(* CoDeSys 2.3 library: Flexlink V2_0.lib *)
(* Libraries: TcUtilities.lib*3.2.16 16:08:58, TcSystem.lib*24.2.16 14:35:18, TcBase.lib 14.5.09 12:14:08, STANDARD.LIB 5.6.98 12:03:02, TcEtherCAT.lib 1.12.15 17:38:26 *)

(* Global variable list: Global_Variables *)
VAR_GLOBAL
(**************************************************************************************************************)
(* System Bit *)
(**************************************************************************************************************)

	OFF_50ms		: BOOL;
	ON_50ms		: BOOL;
	Clock50msOnPls	: BOOL;
	OFF_100ms		: BOOL;
	ON_100ms		: BOOL;
	Clock100msOnPls	: BOOL;
	OFF_500ms		: BOOL;
	ON_500ms		: BOOL;
	Clock500msOnPls	: BOOL;
	OFF_1s			: BOOL;
	ON_1s			: BOOL;
	Clock1sOnPls	: BOOL;
	Always_ON		:BOOL;
	Always_Off		:BOOL;
	Debug			:BOOL := TRUE;

(**************************************************************************************************************)
(* Machine Standard Word *)
(**************************************************************************************************************)

	ErrorDWord 			AT %MD1000:  ARRAY [0..20,1..10] OF DWORD;
	WarningDWord		AT%MD2000: ARRAY [0..20,1..10] OF DWORD;
	AutoDWord 			AT %MD3000:  ARRAY [0..20,1..10] OF DWORD;
	OriginDWord 			AT %MD4000:  ARRAY [0..20,1..10] OF DWORD;

	InputByte				AT %IB0: ARRAY [0..500] OF BYTE;
	OutputByte			AT %QB0: ARRAY [0..500] OF BYTE;

(**************************************************************************************************************)
(* Machine and Station Control *)
(**************************************************************************************************************)
	MC:Struc_Machine_Ctrl;
	SC :ARRAY[0..20] OF Struc_Station_Ctrl;

(**************************************************************************************************************)
(* Manual Control *)
(**************************************************************************************************************)
	ManualSafetyOK		:BOOL;
	M_StepFwdPls		:BOOL;
	M_StepBwdPls		:BOOL;
	M_StepRun			:BOOL;

(**************************************************************************************************************)
(* Input/Output *)
(**************************************************************************************************************)
	InputWord			AT%IB0	:ARRAY [0..100] OF BOOL;


END_VAR

(* Global variable list: Global_Variables_Error *)
VAR_GLOBAL
	E_EmgStop			: BOOL;
	E_LightCurtain		: BOOL;
	E_AirLow 			: BOOL;
	E_SafetyDoorOpen	: BOOL;
END_VAR

(* Global variable list: Global_Variables_HMI *)
VAR_GLOBAL
	T_AutoRunString:		STRING;

	T_StepRun:			BOOL;
	T_StepStop:			BOOL;
	T_StepBwd:			BOOL;
	T_StepFwd:			BOOL;
	T_StationError:		BOOL;
	T_Origin:				BOOL;
	T_OneCycleRun:		BOOL;
	T_ManualCycleTime:	TIME;
	T_Curr_Step_Station: 	UINT;
	T_EndProd:			BOOL;

	V_StepRunCurrStation:	STRING;
	V_StepRunStatus:		STRING;
	V_AutorunString:		STRING;
END_VAR

(* Global variable list: Global_Variables_Holding *)
VAR_GLOBAL RETAIN
	Password_Control: Std_Password_Ctrl;

(* Parameter Setting *)
	Number_of_Station : INT;

END_VAR

(* Data type *)
TYPE E_IndradriveDriveState :
(
	DriveState_Mode_PM  := 0,
	DriveState_Mode_bb,
	DriveState_Mode_Ab,
	DriveState_Mode_AH,
	DriveState_Mode_AF,
	DriveState_Mode_FC,
	DriveState_Mode_PC,
	DriveState_Mode_Invalid
);
END_TYPE

(* Data type *)
TYPE E_IndradriveErrorCode :
(
	INDRADRIVE_NO_ERROR := 0,
	INDRADRIVE_INVALID_ADDRESS_VALUE,
	INDRADRIVE_INVALID_DATA_VALUE,
	INDRADRIVE_PARA_WRITE_ERROR,
	INDRADRIVE_PARA_READ_ERROR,

	INDRADRIVE_ERROR_UNKNOWN := 999
);
END_TYPE

(* Data type *)
TYPE E_IndradriveListIndex :
(
	LIST_INDEX_0  := 0,
	LIST_INDEX_1,
	LIST_INDEX_2,
	LIST_INDEX_3,
	LIST_INDEX_4,
	LIST_INDEX_5,
	LIST_INDEX_6,
	LIST_INDEX_7,
	LIST_INDEX_8,
	LIST_INDEX_9,
	LIST_INDEX_10,
	LIST_INDEX_11,
	LIST_INDEX_12,
	LIST_INDEX_13,
	LIST_INDEX_14,
	LIST_INDEX_15,
	LIST_INDEX_16,
	LIST_INDEX_17,
	LIST_INDEX_18,
	LIST_INDEX_19,
	LIST_INDEX_20,
	LIST_INDEX_21,
	LIST_INDEX_22,
	LIST_INDEX_23,
	LIST_INDEX_24,
	LIST_INDEX_25,
	LIST_INDEX_26,
	LIST_INDEX_27,
	LIST_INDEX_28,
	LIST_INDEX_29,
	LIST_INDEX_30,
	LIST_INDEX_31,
	LIST_INDEX_MAX
);
END_TYPE

(* Data type *)
TYPE E_IndradriveOpMode :
(
	OP_MODE_DCP  := 0,
	OP_MODE_POS_01,
	OP_MODE_MUX_01,
	OP_MODE_MUX_02,
	OP_MODE_PROCESS_CNTRL,
	OP_MODE_USER := 99
);
END_TYPE

(* Data type *)
TYPE ST_ChecksumConfig :
STRUCT
	arChecksumConfigList            :  ARRAY [0..LIST_INDEX_MAX] OF WORD;       (* Read / write S_0_0327, IDN list of checksum parameter *)
	wCheckSumExpected             : WORD;                                                                     (* Read / write S-0-0326, Parameter checksum *)
END_STRUCT
END_TYPE

(* Data type *)
TYPE st_Indradrive_DCP_input :
STRUCT
	wAntriebsstatuswort   			: WORD;
	wSignalstatuswort   			: WORD;
	diLageistwert		  			: DINT;
	diIstgeschwindigkeit  			: DINT;
	dwDiagnosenummer				: DWORD;
END_STRUCT
END_TYPE

(* Data type *)
TYPE st_Indradrive_DCP_output :
STRUCT
	wMastersteuerwort   			: WORD;
	wSignalsteuerwort   			: WORD;
	diPositioniersollwert  			: DINT;
	diPositioniergeschwindigkeit  	: DINT;
END_STRUCT
END_TYPE

(* Data type *)
TYPE st_Indradrive_DCP_using_MUX_8_input :
STRUCT
	wDriveStatusWord : WORD;        (* S-0-0135: Drive Status word*)
	stMUX_in                 : st_Indradrive_MUX_8_input; (* 8 Channel Multiplexer Input Structure *)
END_STRUCT
END_TYPE

(* Data type *)
TYPE st_Indradrive_DCP_using_MUX_8_output :
STRUCT
	wMasterControlWord  : WORD;        (* S-0-0134: Master Control Word*)
	stMUX_out               : st_Indradrive_MUX_8_output; (* 8 Channel Multiplexer Output Structure *)
END_STRUCT
END_TYPE

(* Data type *)
TYPE st_Indradrive_MUX_1_input :
STRUCT
(*Struktur der benötigten Multiplexparameter (Teil der Echtzeitkanal-Eingangsdaten*)
	uiIndexAdressing	: UINT;		(*S-0-0368*)
      	uiListIndexWrite		: UINT;		(*S-0-0362*)
      	uiListIndexRead		: UINT;		(*S-0-0366*)
      	diReadValue1		: DINT;		(*S-0-0364*)
END_STRUCT
END_TYPE

(* Data type *)
TYPE st_Indradrive_MUX_1_output :
STRUCT
(*Struktur der benötigten Multiplexparameter (Teil der Echtzeitkanal-Ausgangsdaten*)
	uiIndexAdressing		: UINT;		(*S-0-0368*)
	uiListIndexWrite		: UINT;		(*S-0-0362*)
       	uiListIndexRead		: UINT;		(*S-0-0366*)
       	diWriteValue1		: DINT;		(*S-0-0360*)
END_STRUCT
END_TYPE

(* Data type *)
TYPE st_Indradrive_MUX_8_input :
STRUCT
(*Struktur der benötigten Multiplexparameter (Teil der Echtzeitkanal-Eingangsdaten*)
	uiIndexAdressing	: UINT;            (*S-0-0368*)
      	uiListIndexWrite		: UINT;            (*S-0-0362*)
      	uiListIndexRead		: UINT;            (*S-0-0366*)
      	dwReadValue1		: DWORD;     (*S-0-0364*)
    	dwReadValue2 		: DWORD;     (*S-0-0480 *)
    	dwReadValue3 		: DWORD;     (*S-0-0481 *)
    	dwReadValue4 		: DWORD;     (*S-0-0482 *)
    	dwReadValue5 		: DWORD;     (*S-0-0483 *)
    	dwReadValue6 		: DWORD;     (*S-0-0484 *)
    	dwReadValue7 		: DWORD;     (*S-0-0485 *)
    	dwReadValue8 		: DWORD;     (*S-0-0486 *)
END_STRUCT
END_TYPE

(* Data type *)
TYPE st_Indradrive_MUX_8_output :
STRUCT
(*Struktur der benötigten Multiplexparameter (Teil der Echtzeitkanal-Ausgangsdaten*)
	uiIndexAdressing		 : UINT;		    (*S-0-0368*)
	uiListIndexWrite		        : UINT;		    (*S-0-0362*)
     	uiListIndexRead		        : UINT;		    (*S-0-0366*)
      	dwWriteValue1                 : DWORD;      (*S-0-0360*)
	dwWriteValue2                 : DWORD;      (*S-0-0450 *)
	dwWriteValue3                 : DWORD;      (*S-0-0451 *)
	dwWriteValue4                 : DWORD;      (*S-0-0452 *)
	dwWriteValue5                 : DWORD;      (*S-0-0453 *)
	dwWriteValue6                 : DWORD;      (*S-0-0454 *)
	dwWriteValue7                 : DWORD;      (*S-0-0455 *)
	dwWriteValue8                 : DWORD;      (*S-0-0456 *)
END_STRUCT
END_TYPE

(* Data type *)
TYPE st_Indradrive_ProcessControl_input :
STRUCT
	wDriveStatusWord : WORD;                                                  (* S-0-0135: Drive Status word*)
	wSignalStatusWord : WORD;                                                (* S-0-0144: Singal Status word*)
	wProcessControlStatusWord : WORD;                              (* P-0-1410: Process Control status word coming from MLD program*)
	diVelocityAct : DINT;                                                                 (* S-0-0040: Actual velocity *)
	diPressureAct : DWORD;                                                               (* P-0-1372: Actual pressure value coming from MLD program  *)
	wAxisControllerMessage : WORD;                                      (*P-0-0555: Axis Controller Messages *)
	dwDriveDiagnosticNumber : DWORD;                               (* S-0-0390: Drive Diagnostic number *)
	diFlowAct :DWORD; 							    (* S-0-1301: Actual flow *)
	diAxisControllerMessage:WORD; 				    (*P-0-0555 Axis controller message*)
END_STRUCT
END_TYPE

(* Data type *)
TYPE st_Indradrive_ProcessControl_MUX_input :
STRUCT
	wDriveStatusWord : WORD;        (* S-0-0135: Drive Status word*)
	stMUX_in                 : st_Indradrive_MUX_8_input; (* 8 Channel Multiplexer Input Structure *)
END_STRUCT
END_TYPE

(* Data type *)
TYPE st_Indradrive_ProcessControl_MUX_output :
STRUCT
	wMasterControlWord  : WORD;        (* S-0-0134: Master Control Word*)
	stMUX_out               : st_Indradrive_MUX_8_output; (* 8 Channel Multiplexer Output Structure *)
END_STRUCT
END_TYPE

(* Data type *)
TYPE st_Indradrive_ProcessControl_output :
STRUCT
	wMasterControlWord  : WORD;          (* S-0-0134: Master Control Word*)
	wSignalControlWord : WORD;            (* S-0-0145: Signal Control Word*)
	wProcessControlWord : WORD;        (* P-0-1390: Process Control, Control Word, going to MLD Program *)
	diVelocityCmd : DINT;                            (* S-0-0036: Velocity Command value *)
	diPressureCmd : DINT;                          (* P-0-1371:Pressure Command value going to MLD Program *)
	diVolumePump01:DWORD; (**)
	diVolumePump02:DWORD;
	diVelocityLimitPos : DINT;                     (* P-0-1377:Postive Velocity Limit going to MLD Program *)
END_STRUCT
END_TYPE

(* Data type *)
TYPE Struc_Hist_Step_Case :
STRUCT
	CurrentStepHist	: INT;
	NextStepHist		: INT;
	StepTime		: TIME;
END_STRUCT
END_TYPE

(* Data type *)
TYPE Struc_Machine_Ctrl :
STRUCT
(* Mode Bit*)
	AutoMode		:BOOL;
	ManualMode		:BOOL;

(* Status Bit*)
	DryRun			:BOOL;
	Stop			:BOOL;
	AutoRunning		:BOOL;
	StopPressed		:BOOL;


	StationStopErr 	:BOOL;
	Warning			:BOOL;
	WarningBuzzer	:BOOL;
	Trouble			:BOOL;
	ErrDetection		:BOOL;


	OriginSchRun		:BOOL;
	InxOrigin			:BOOL;
	AllOrigin			:BOOL;
	AllStationRdy		:BOOL;
	AllStationNoWP 	:BOOL;

END_STRUCT
END_TYPE

(* Data type *)
TYPE Struc_Station_Ctrl :
STRUCT

	Running			:BOOL;
	AutoRun			:BOOL;
	RunReq			:BOOL;		(*Station Start Work Request*)
	Done			:BOOL;		(*Station Work Complete*)
	RunCond		:BOOL;
	Run_NextStepPls	:BOOL;
	Run_PrevStepPls	:BOOL;
	M_Step			:BOOL;

	Origin			:BOOL;   		(* Station Already Origin *)
	Rdy				:BOOL;		(* Station Ready *)
	NoWP 			:BOOL;
	MajorFault		:BOOL;		(* Station Major Fault *)
	MinorFault		:BOOL;		(* Station Minor Fault *)
	Warning			:BOOL;		(* Station Warning *)
	Bypass			:BOOL;		(* Station Bypass *)
	OriginSchRun		:BOOL;		(* Request Station to Origin *)

	Name			:STRING;
	Status			:STRING;
	CycleTime		:TIME;

END_STRUCT
END_TYPE

(* Data type *)
TYPE structIndradrive :
STRUCT
	In_ServoOn:BOOL;
	In_JogFwd:BOOL;
	In_JogBwd:BOOL;
	In_MoveHome:BOOL;
	In_SetAbsRef:BOOL;
	In_MoveAbs:BOOL;
	In_MoveRel:BOOL;
	In_StopMove:BOOL;
	In_VelCmd:REAL;
	In_PosCmd:REAL;
	In_MoveXLock:BOOL;	(*Mechanical Interlock*)
	Out_Ready:BOOL;
	Out_Busy:BOOL;
	Out_InPos:BOOL;
	Out_Referenced:BOOL;
	Out_PosLimit:BOOL;	(*1=OK*)
	Out_NegLimit:BOOL;	(*1=OK*)
	Out_Error:BOOL;
	Out_Warning:BOOL;
	Out_ErrorWord:WORD;
	Out_CurrPos:REAL;
	Out_CurrVel:REAL;
	Out_PosDirc:BOOL;	(*Moving in Positive Direction*)
	Out_NegDirc:BOOL;	(*Moving in Negative Direction*)
END_STRUCT
END_TYPE

(* POU Password_Output, ST *)
PROGRAM Password_Output
VAR

	pls_PasswordOK: R_TRIG;
	PasswordOKPls:BOOL;
END_VAR
(**************************************************************************************************************)
(* HMI Password Control*)
(**************************************************************************************************************)

Password_Control(
	In_PasswordConfig:= '9999');

pls_PasswordOK(CLK:= Password_Control.Out_PasswordOK OR Password_Control.Out_PasswordChanged);
PasswordOKPls := pls_PasswordOK.Q;

IF PasswordOKPls THEN
	CurrentVisu := 'TP40_SETTING';
END_IF
END_PROGRAM

(* POU Std_System_Out, LD *)
PROGRAM Std_System_Out
VAR

	Clk50ms:TON;
	ClkOff50ms:TON;
	Clk100ms:TON;
	ClkOff100ms:TON;
	Clk500ms:TON;
	ClkOff500ms:TON;
	ClkOn1s:TON;
	ClkOff1s:TON;

	T50ms_RTRIG: R_TRIG;
	T100ms_RTRIG: R_TRIG;
	T500ms_RTRIG: R_TRIG;
	T1s_RTRIG: R_TRIG;

END_VAR
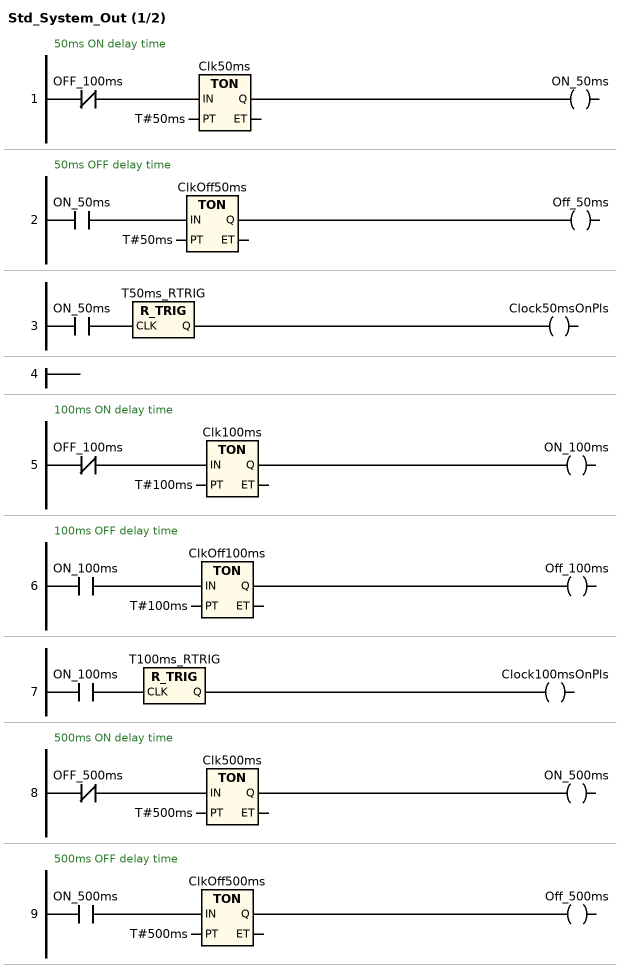
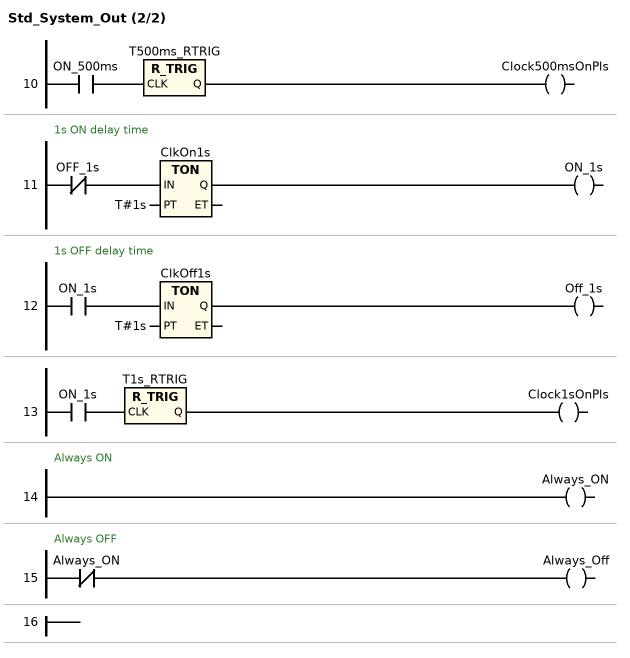
_LD_ (* Ladder Diagram *)
NETWORK 1 (* 50ms ON delay time *)
	[/OFF_100ms] - Clk50ms:TON(IN: *, PT: T#50ms) --- (ON_50ms)
NETWORK 2 (* 50ms OFF delay time *)
	[ON_50ms] - ClkOff50ms:TON(IN: *, PT: T#50ms) --- (Off_50ms)
NETWORK 3
	[ON_50ms] - T50ms_RTRIG:R_TRIG(CLK: *) --- (Clock50msOnPls)
NETWORK 4
	*
NETWORK 5 (* 100ms ON delay time *)
	[/OFF_100ms] - Clk100ms:TON(IN: *, PT: T#100ms) --- (ON_100ms)
NETWORK 6 (* 100ms OFF delay time *)
	[ON_100ms] - ClkOff100ms:TON(IN: *, PT: T#100ms) --- (Off_100ms)
NETWORK 7
	[ON_100ms] - T100ms_RTRIG:R_TRIG(CLK: *) --- (Clock100msOnPls)
NETWORK 8 (* 500ms ON delay time *)
	[/OFF_500ms] - Clk500ms:TON(IN: *, PT: T#500ms) --- (ON_500ms)
NETWORK 9 (* 500ms OFF delay time *)
	[ON_500ms] - ClkOff500ms:TON(IN: *, PT: T#500ms) --- (Off_500ms)
NETWORK 10
	[ON_500ms] - T500ms_RTRIG:R_TRIG(CLK: *) --- (Clock500msOnPls)
NETWORK 11 (* 1s ON delay time *)
	[/OFF_1s] - ClkOn1s:TON(IN: *, PT: T#1s) --- (ON_1s)
NETWORK 12 (* 1s OFF delay time *)
	[ON_1s] - ClkOff1s:TON(IN: *, PT: T#1s) --- (Off_1s)
NETWORK 13
	[ON_1s] - T1s_RTRIG:R_TRIG(CLK: *) --- (Clock1sOnPls)
NETWORK 14 (* Always ON *)
	* --- (Always_ON)
NETWORK 15 (* Always OFF *)
	[/Always_ON] --- (Always_Off)
NETWORK 16
	*
_END_LD_
(* the same logic as Structured Text *)
(* Network 1: 50ms ON delay time *)
Clk50ms(IN := NOT OFF_100ms, PT := T#50ms);
ON_50ms := Clk50ms.Q;
(* Network 2: 50ms OFF delay time *)
ClkOff50ms(IN := ON_50ms, PT := T#50ms);
Off_50ms := ClkOff50ms.Q;
(* Network 3 *)
T50ms_RTRIG(CLK := ON_50ms);
Clock50msOnPls := T50ms_RTRIG.Q;
(* Network 4 *)
(* Network 5: 100ms ON delay time *)
Clk100ms(IN := NOT OFF_100ms, PT := T#100ms);
ON_100ms := Clk100ms.Q;
(* Network 6: 100ms OFF delay time *)
ClkOff100ms(IN := ON_100ms, PT := T#100ms);
Off_100ms := ClkOff100ms.Q;
(* Network 7 *)
T100ms_RTRIG(CLK := ON_100ms);
Clock100msOnPls := T100ms_RTRIG.Q;
(* Network 8: 500ms ON delay time *)
Clk500ms(IN := NOT OFF_500ms, PT := T#500ms);
ON_500ms := Clk500ms.Q;
(* Network 9: 500ms OFF delay time *)
ClkOff500ms(IN := ON_500ms, PT := T#500ms);
Off_500ms := ClkOff500ms.Q;
(* Network 10 *)
T500ms_RTRIG(CLK := ON_500ms);
Clock500msOnPls := T500ms_RTRIG.Q;
(* Network 11: 1s ON delay time *)
ClkOn1s(IN := NOT OFF_1s, PT := T#1s);
ON_1s := ClkOn1s.Q;
(* Network 12: 1s OFF delay time *)
ClkOff1s(IN := ON_1s, PT := T#1s);
Off_1s := ClkOff1s.Q;
(* Network 13 *)
T1s_RTRIG(CLK := ON_1s);
Clock1sOnPls := T1s_RTRIG.Q;
(* Network 14: Always ON *)
Always_ON := TRUE;
(* Network 15: Always OFF *)
Always_Off := NOT Always_ON;
(* Network 16 *)
END_PROGRAM

(* POU F_GetVersionDC_IA_Indradrive, ST *)
FUNCTION F_GetVersionDC_IA_Indradrive : UINT
VAR_INPUT
       nVersionElement       :       INT;
END_VAR 
VAR
END_VAR
(* Version history:
Date               | Version  | created under             | Author            | Remark 
------------------------------------------------------------------------------------------------------------------------------------------------------------------------------ 
03/01/2012    | 1.0.0      | V2.11.0 (Build 1514) | U. Chauhan   | first release 
------------------------------------------------------------------------------------------------------------------------------------------------------------------------------ 
20/08/2012    | 1.1.0      | V2.11.0 (Build 1514) | U. Chauhan   | 
	Old Process Control FB is renamed as Process control using MUX Version 1.0. 
	New ProcessControl FB Version 1.0 without MUX added.
------------------------------------------------------------------------------------------------------------------------------------------------------------------------------ 
29/10/2012    | 1.1.1      | V2.11.0 (Build 1514) | U. Chauhan   | "Process Control FB" and "Process control using MUX FB"  updated to Version 1.1
	DriveAH Bit added to both the FB and activated along with DriveStart Input.
11/12/2012    | 1.1.2      | V2.11.0 (Build 1514) | U. Chauhan   | "Process Control FB" updated to Version 1.2 and "Process control using MUX FB" updated to Version 1.2
	some bug fixes and calculations updated as per  
18/02/2013    | 1.2.0      | V2.11.0 (Build 1514) | U. Chauhan   | "Process Control FB" updated to Version 1.3 
	It is now possibile to use Pressure Value and Flowrate values in Percentage, 
	Selection of the Parameter Set is now possible with Input field
	FlowRateMaximum vlaue will be passed on to Drive as a positive Velocity Limit
05/08/2013    | 1.3.0      | V2.11.0 (Build 1514) | U. Chauhan   | SIP Implementation for Parameter Access added.
					FBs for Read Everything, ReadDescription, ReadOnlyData, ReadSegment, Read DataStatus,
					WriteData and WriteDatabits added.
------------------------------------------------------------------------------------------------------------------------------------------------------------------------------ 
26/02/2014    | 2.0.0      | V2.11.0 (Build 1514) | U. Chauhan   | SIPParameter Access FBs have been moved to another library due to license issues with TCPIP server. 
------------------------------------------------------------------------------------------------------------------------------------------------------------------------------ 
20.08.2014     |2.1.0	     | V2.11.0 (Build 1514) | Arun R            | FB_ProcessControl update of drive halt and flow rate decimal point logic. 
------------------------------------------------------------------------------------------------------------------------------------------------------------------------------ 
15/09/2014     |2.2.0	     | V2.11.0 (Build 1514) | Pradeep R           |  FB_Indradrive_DCP drive enable updated to stay on always to prevent torque free mode 
------------------------------------------------------------------------------------------------------------------------------------------------------------------------------ 
*) 

CASE nVersionElement OF
1: (* major number *)
       F_GetVersionDC_IA_Indradrive := 2;
2: (* minor number *)
       F_GetVersionDC_IA_Indradrive := 2;
3: (* revision number *)
       F_GetVersionDC_IA_Indradrive := 0;
ELSE
   F_GetVersionDC_IA_Indradrive := 16#FFFF;
END_CASE
END_FUNCTION

(* POU FB_ConfigChecksum, ST *)
(*#########################################################################################*)
(* General Header *)
(*----------------------------------------------------------------------------------------------------------------------------------------------------------------*)
(* Short description :		      Function Block for configuring & checking Checksum parameters in Indradrive              *)
(* Version : 					      01VRS                                                                                                                                       *)
(* Name : 					      Upendra Chauhan                                                                                                                    *)
(* Date : 					      2012-03-23                                                                                                                               *)
(* Company : 				      Bosch Rexroth AG                                                                                                                    *)
(* Target : 					      >MPx07VRS                                                                                                                             *)
(* Functional description :		With the help of this function block configurable Checksum feature of Indradrive            *)
(*                                                     User defined parameter list is at first written to paramter S-0-0327                            *)
(*                                                     This is enable the drive to calculate the checksum value for these parameter which is  *)
(*                                                     in turn written by Indradrive to Parameter S-0-0326                                                            *)
(*                                                     The FB reads this parameter anc compare is with Desired Checksum value as given *)
(*                                                     by user. If the value match the desired checksum good result is stored in  output           *)
(*                                                     bCheckSumOk. Actual checksum value is stored in dwActCheckSum and error Id is   *)
(*                                                     displayed in case of any error in dwErrorID                                                                         *)
(*----------------------------------------------------------------------------------------------------------------------------------------------------------------*)
(* Handling specials :                                                                                                                                                                      *)
(*----------------------------------------------------------------------------------------------------------------------------------------------------------------*)
(* Additional Header                                                                                                                                                                        *)
(*----------------------------------------------------------------------------------------------------------------------------------------------------------------*)
(* Version : 					 *)
(* Name : 					 *)
(* Date : 						 *)
(* Company : 					 *)
(* *)
(* *)
(* *)
(*-----------------------------------------------------------------------------------------------------------------------------------------------------------------*)
(*##########################################################################################*)
(*##########################################################################################*)
FUNCTION_BLOCK FB_ConfigChecksum
VAR_INPUT
	bExecute			 : BOOL;
	pstPlcDriveRef          : POINTER TO ST_PLCDriveRef;
	pstChecksumConfig : POINTER TO ST_ChecksumConfig;
END_VAR
(*___________________________________________________________________________________________________________________*)
(*___________________________________________________________________________________________________________________*)
VAR_OUTPUT
	bActive				: BOOL;										(*FB Active*)
	bDone                       : BOOL;
	bError				: BOOL;										(*Error in FB*)
	bCheckSumOk		: BOOL;										(*TRUE - Right config loaded / FALSE- Wrong Config*)
	dwActCheckSum     : DWORD := 0;                                                          (* Actual Checksum value, S-0-0326, Parameter checksum *)
	dwErrorID                 : DWORD := 0;                                                          (* Actual Checksum value, S-0-0326, Parameter checksum *)
END_VAR

VAR_IN_OUT
END_VAR
(*___________________________________________________________________________________________________________________*)
(*___________________________________________________________________________________________________________________*)
VAR
	stDriveRef                 : ST_DriveRef;
	iStep				: USINT;
	nElement 			: BYTE 				:=  64 ;					(*In case of list parameter the element of the list to be read or written*)
	bReadPar      		: BOOL 			:= FALSE;				(*command to read the parameter*)
	bReadErr       		: BOOL;										(*error in reading*)
	bWritePar			: BOOL;										(*command to write the parameter*)
	bWriteActive		: BOOL;										(*writing in progress*)
	bErrorWrite			: BOOL;										(*error in writing*)
	bWriteErr			: BOOL;										(*error in writing*)
	bReadActive		: BOOL;										(*reading in progress*)


	arConfigByteValue 	: ARRAY [0..100] OF BYTE;		     			(*array of bite values*)

 	 (*Function block declaration*)
	fbSercosParaWrite	: FB_SoEWrite_ByDriveRef;				(*write fb call*)
	fbSercosParaRead	: FB_SoERead_ByDriveRef;				(*read fb call*)
(*___________________________________________________________________________________________________________________*)
	iListIndex : INT := 0;
	wNoOfBytesTransfered: WORD;
	arbyReadValue : ARRAY [0..4] OF BYTE;
	R_TRIG_bExecute: R_TRIG;
END_VAR
(*___________________________________________________________________________________________________________________
Name of the Project			:CheckSumFBCode.pro
Name of the PLC System		:TWINCAT
Name of the DRIVE/Firmware	:Rexroth Indradrive HCS01.1E / 16VRS 
Version of Software used		:TwinCAT V2.11.0(Build 2209)
Version of Function Block		:V1.0
Author						: Upendra Chauhan
Date						:23.03.2012
___________________________________________________________________________________________________________________*)

(*FUNCTION BLOCK USED TO VERIFY THE CONFIGURATION FOR REXROTH INDRA DRIVE SETTINS ARE MADE CORRECTLY*)

(* rising edge at bExecute *)
R_TRIG_bExecute ( CLK := bExecute );

(* execute cycle *)
CASE iStep OF
	0:										(*WAIT FOR EXECUTE COMMAND*)
		 IF R_TRIG_bExecute.Q THEN
			bActive :=TRUE;
			dwActCheckSum := 0;                                                          (* Actual Checksum value, S-0-0326, Parameter checksum *)
			iStep:=1;
		 END_IF

		IF (bExecute = FALSE) THEN
			bDone :=FALSE;
			bError := FALSE;
			bCheckSumOk :=FALSE;
			dwErrorID := INDRADRIVE_NO_ERROR;
		 END_IF

	1:
		IF pstPlcDriveRef = 0 OR pstChecksumConfig = 0 THEN
			dwErrorID := INDRADRIVE_INVALID_ADDRESS_VALUE;
			iStep:=200;
		ELSE
			iStep:=5;
		END_IF

	5:
		stDriveRef.sNetId     := F_CreateAmsNetId(pstPlcDriveRef^.aNetId);
		stDriveRef.nSlaveAddr := pstPlcDriveRef^.nSlaveAddr;
		stDriveRef.nDriveNo   := pstPlcDriveRef^.nDriveNo;
		stDriveRef.nDriveType := pstPlcDriveRef^.nDriveType;
		IF (stDriveRef.sNetId <> '') AND (stDriveRef.nSlaveAddr <> 0) THEN
			iStep:= 10;
		ELSE
			dwErrorID := INDRADRIVE_INVALID_DATA_VALUE;
			iStep:= 200;
		END_IF

	10:
		FOR iListIndex := 0 TO LIST_INDEX_MAX DO
			IF  ( pstChecksumConfig^.arChecksumConfigList[iListIndex] = 0 )
			THEN
				IF iListIndex = 0 THEN
					(* if First two parameter are Zero then error exit *)
					IF ( pstChecksumConfig^.arChecksumConfigList[iListIndex + 1] = 0 ) THEN
						dwErrorID := INDRADRIVE_INVALID_DATA_VALUE;
						iStep:= 200;
						(* exit loop as list has invalid *)
						EXIT;
					END_IF
				ELSE
					(* if two consicutive parameter are Zero or Last list para is zero , the list is completed *)
					IF ( pstChecksumConfig^.arChecksumConfigList [iListIndex -1] = 0 ) OR
					    (  iListIndex = LIST_INDEX_MAX )
					THEN
						IF ( pstChecksumConfig^.arChecksumConfigList [iListIndex -1] = 0 )
						THEN
							(* reduce one step if last value was also zero *)
							iListIndex := iListIndex - 1;
						END_IF
						(* exit loop as list is completed *)
						EXIT;
					END_IF
				END_IF
			END_IF
		END_FOR

		(* Byte length = Number of words x 2 *)
		wNoOfBytesTransfered :=  iListIndex  * 2 ;

		(* first four values of arConfigByteValue depends on the number of Bytes to be transfered *)
		(* convert word value Maximum bytes to array of bytes *)
		MEMCPY ( ADR(arConfigByteValue), ADR(wNoOfBytesTransfered ), 2);
		(* convert word value Maximum bytes to array of bytes *)
		MEMSET ( ADR(arConfigByteValue[2]), 0, 2);
		(* convert wrod array to byte array *)
		MEMCPY ( ADR(arConfigByteValue[4]), ADR(pstChecksumConfig^.arChecksumConfigList), SIZEOF (pstChecksumConfig^.arChecksumConfigList));

		(* write S_0_0327, IDN list of checksum parameter *)
		bWritePar :=TRUE;

		iStep          :=15;

	15:										(*WAIT TILL WRITE bExecuteS*)
		IF bErrorWrite THEN
			(* error writing parameter to Indradrive *)
			dwErrorID := INDRADRIVE_PARA_WRITE_ERROR;
			bWritePar := FALSE;
			iStep:=200;
		ELSE
			IF( NOT bWriteActive ) THEN
				bWritePar := FALSE;
				iStep:=20;
			END_IF
		END_IF

	20:										(*READ THE S326 CHECKSUM VALUE PARAMETER*)
		bReadPar:=TRUE;
		iStep:=25;

	25:										(*WAIT TILL READ bExecuteS*)
		IF bReadErr THEN
			(* error reading parameter from Indradrive *)
			dwErrorID := INDRADRIVE_PARA_READ_ERROR;
			bReadPar:= FALSE;
			iStep:=200;
		ELSE
			IF( NOT bReadActive ) THEN
				bReadPar:= FALSE;
				iStep:=30;
			END_IF
		END_IF

	30:										(*CONVERT READ BYTE VALUE TO WORD VALUE*)
		(* copy read checksum  Byte array to word value *)
		MEMCPY (ADR (dwActCheckSum), ADR(arbyReadValue), 4);
		iStep:=35;

	35:										(*COMPARE WITH PREPROGRAMMED CHECKSUM VALUE TO VALIDATE RIGHT CONFIGURATION*)
		IF ( dwActCheckSum = pstChecksumConfig^.wCheckSumExpected) THEN
			bCheckSumOk :=TRUE;
		ELSE
			bCheckSumOk :=FALSE;
		END_IF
		iStep  :=40;

	40:										(*RESET FUNCTION BLOCK*)
		bDone :=TRUE;
		bActive:=FALSE;
		iStep:=0;

	200:									(*ERROR STEP*)
		bActive:=FALSE;
		bError := TRUE;
		iStep := 0;
END_CASE


(*Write fub function call*)
fbSercosParaWrite(
	stDriveREf := stDriveRef,
	nIdn:= 327 ,                                                            (* Parameter S-0-0327 : IDN list of checksum parameter *)
	nElement:= nElement  ,                                        (* Write 'Value' nElement := 0x40 *)
	pSrcBuf:=ADR (arConfigByteValue) ,
	cbBufLen:=SIZEOF(arConfigByteValue) ,
	bExecute:=bWritePar ,
	tTimeout:=T#10s,
	bBusy=>bWriteActive ,
	bError=>bWriteErr ,
	iAdsErrId=> ,
	 iSercosErrId => );

(*Read fub function call*)
fbSercosParaRead(
	stDriveREf := stDriveRef,
	nIdn:=326 ,                                                            (* Parameter S-0-0326 : checksum value *)
	nElement:=nElement ,                                         (* read 'Value' nElement := 0x40 *)
	pDstBuf:= ADR (arbyReadValue) ,
	cbBufLen:= SIZEOF(arbyReadValue) ,
	bExecute:=bReadPar ,
	tTimeout:=T#10s ,
	bBusy=>bReadActive	 ,
	bError=>bReadErr ,
	iAdsErrId=> ,
	iSercosErrId => ,
	dwAttribute => );
END_FUNCTION_BLOCK

(* POU FB_Indradrive_DCP, ST *)
(*############################################################################################*)
(* General Header *)
(*-----------------------------------------------------------------------------------------------------------------------------------------------------------------*)
(* Short description :			Funktionsbaustein „Antriebsgeführtes Positionieren“ über Ehtercat *)
(* Version : 					01VRS *)
(* Name : 					Michael Lippert *)
(* Date : 						2010-11-12*)
(* Company : 					BoschRexroth AG *)
(* Target : 					>MPx07VRS *)
(* Functional description :		Mit Hilfe dieses Funktionsbausteins „DCP_INDRADRIVE“ kann der Antrieb in der
								Betriebsart „Antriebsgeführtes Positionieren“ durch Vorgabe des S-0-0282,
								Positioniersollwert (POS_CMD) und des S-0-0259, Positioniergeschwindigkeit (VEL_CMD) 
								relativ oder absolut positioniert werden. Mit diesem Funktionsbaustein werden ferner 
								die Funktionen Tippen, Referenzieren und Fehler löschen angesteuert.
*)
(* Handling specials : *)
(*-----------------------------------------------------------------------------------------------------------------------------------------------------------------*)
(* Additional Header *)

(*------------------------------------------------------------------------------------------------------------------------------------------------------------------------*)
(* Version : 1.1.0	                                                                                                                                                                                              *)
(* Name : prd6kor ( DC-IA/EDY )                                                                                                                                                                   *)
(*Date: 15.09.2014                                                                                                                                                                                                *)
(* Company : Bosch Rexroth                                                                                                                                                                            *)
(* "FB_Indradrive_DCP" updated drive enable to prevent torque free mode on motor					                      *)
(*------------------------------------------------------------------------------------------------------------------------------------------------------------------------*)


(*############################################################################################*)
(*############################################################################################*)
FUNCTION_BLOCK FB_Indradrive_DCP
VAR_INPUT
     bDRIVE_ENABLE 					: BOOL; 						(*Antriebstatus Uebergang AB -> AH, Drive Enable state of drive change Ab->AH *)
     bDRIVE_START 					: BOOL; 						(*Antriebstatus Uebergang AH -> AF, Drive Enable state of drive change AH->AF *)
     bHOMING 							: BOOL; 						(*Achse Referenzieren, Homing the axis*)
     bRESET 							: BOOL; 						(*Stoerung quittieren, Reset Error*)
     bJOG_FORWARD 					: BOOL; 						(*Tippen vorwaerts, Jog forward*)
     bJOG_BACKWARD					: BOOL;						(*Tippen rueckwaerts, Jog backward*)
     bNEW_VALUE 						: BOOL; 						(*neuer Sollwert, new value *)
     bABS_REL 						: BOOL; 						(*Position Absolut = 0 oder Relativ = 1, position = absoluteor relative  *)
     bIMMEDIATE_CHANGE 				: BOOL; 						(*Satzsofortwechsel 1= sofort, immediate block change 1= immediately*)
     diPOS_CMD 						: DINT; 						(*Soll-Position, Command position*)
     diVEL_CMD 						: DINT; 						(*Soll-Geschwindigkeit, command velocity*)
     stEK_IN							: st_Indradrive_DCP_input;		(*Eingangsdaten (input data*)
END_VAR
VAR_OUTPUT
     bQ_DRIVE_ENABLE 				: BOOL; 						(*Quittierung DRIVE_ENABLE, acknowledge DRIVE_ENABLE*)
     bQ_MAIN_MODE 					: BOOL; 						(*Quittierung MAIN_MODE, acknowledge MAIN_MODE*)
     bIN_REFERENCE 					: BOOL; 						(*Referenziert, In_Reference*)
     bPOS_OK 							: BOOL; 						(*Sollwert erreicht = 1, target position reached = 1*)
     bNEW_VALUE_POSSIBLE 			: BOOL; 						(*Neuer Sollwert moeglich, NEW_VALUE_POSSIBLE*)
     bSTATUS_MESSAGE 				: BOOL; 						(*STATUS_MESSAGE*)
     bWARNING 						: BOOL; 						(*WARNING*)
     bERROR 							: BOOL; 						(*ERROR*)
     bIN_STANDSTILL 					: BOOL; 						(*IN_STANDSTILL*)
     dwDRIVE_DIAGNOSIS 				: DWORD; 					(*DRIVE_DIAGNOSIS*)
     diPOS_ACT 						: DINT; 						(*Aktuelle Position, actual position*)
     diVEL_ACT 						: DINT; 						(*Aktuelle Geschwindigkeit, actual velocity*)
     stEK_OUT 							: st_Indradrive_DCP_output;	(*Ausgangsdaten (output data*)
END_VAR
VAR
	bInternHalt 						: BOOL; 						(*INTERN_Halt*)
	bInternFrg 						: BOOL; 						(*INTERN_FRG*)
	bInternPosStart 					: BOOL; 						(*INTERN_POS_START*)
	bInternHoming 					: BOOL; 						(*INTERN_HOMING*)
	bInternJogForward 				: BOOL;						(*INTERN_JOG_FORWARD*)
	bInternJogBackward 				: BOOL; 						(*INTERN_JOG_BACKWARD*)
	bNewValueFlanke 				: BOOL; 						(*NEW_VALUE_FLANKE*)
	bNewValueImpulse 				: BOOL; 						(*NEW_VALUE_IMPULSE*)
END_VAR
(*###############################################################################*)
(*####  Bildung Statusbits Baustein									    	  ###*)
(*###############################################################################*)

(* Drive in AF? *)
bQ_DRIVE_ENABLE				:= stEK_IN.wAntriebsstatuswort.14
									AND stEK_IN.wAntriebsstatuswort.15;

(* Drive enabled (in AF) + Drive Follows Cmd + Primary OpMode active *)
bQ_MAIN_MODE 					:= stEK_IN.wAntriebsstatuswort.3
									AND bQ_DRIVE_ENABLE
									AND NOT stEK_IN.wAntriebsstatuswort.8
									AND NOT stEK_IN.wAntriebsstatuswort.9
									AND NOT stEK_IN.wAntriebsstatuswort.10;

bNEW_VALUE_POSSIBLE			:=   	stEK_OUT.wSignalsteuerwort.0 AND
									 stEK_IN.wSignalstatuswort.10 OR
									(
										NOT stEK_OUT.wSignalsteuerwort.0 AND
										NOT stEK_IN.wSignalstatuswort.10
									) AND
									stEK_IN.wAntriebsstatuswort.15 AND  (* actually redundant with bQ_MAIN_MODE *)
									bQ_MAIN_MODE AND
									bInternPosStart;

(*##################################################################################*)
(*####  Bildung interner Zuständsbits 											 ###*)
(*##################################################################################*)

bInternHoming 					:= bInternFrg AND NOT bInternPosStart AND NOT bJOG_FORWARD
									AND NOT bJOG_BACKWARD AND bHOMING;

bInternJogForward 				:= bInternFrg AND NOT bInternPosStart AND bJOG_FORWARD
									AND NOT bJOG_BACKWARD AND NOT bHOMING;

bInternJogBackward 				:= bInternFrg AND NOT bInternPosStart AND NOT bJOG_FORWARD
									AND bJOG_BACKWARD AND NOT bHOMING;

bInternPosStart					:= bInternFrg AND NOT bJOG_FORWARD
									AND NOT bJOG_BACKWARD AND NOT bHOMING;

bInternHalt						:= bDRIVE_ENABLE;

bInternFrg 						:= bInternHalt AND bQ_DRIVE_ENABLE AND bDRIVE_START;

(*##################################################################################*)
(*####  Bildung Togglebit für Sollwertübernahme 								 ###*)
(*##################################################################################*)

bNewValueImpulse				:= bNEW_VALUE AND NOT bNewValueFlanke;

bNewValueFlanke					:= bNEW_VALUE;

IF (bNEW_VALUE_POSSIBLE OR bIMMEDIATE_CHANGE) AND bInternPosStart AND bNewValueImpulse THEN
	stEK_OUT.diPositioniersollwert := diPOS_CMD;
	IF (stEK_IN.wSignalstatuswort.10 XOR stEK_OUT.wSignalsteuerwort.0) AND bIMMEDIATE_CHANGE THEN
		stEK_OUT.wSignalsteuerwort.0 := stEK_IN.wSignalstatuswort.10;
	ELSE
		stEK_OUT.wSignalsteuerwort.0 := NOT stEK_IN.wSignalstatuswort.10;
	END_IF
(*Verhinderung F2050 -->nicht nötig Anwenderfehler sollen zu Antriebsfehlern führen*)
(*ELSE
	IF stEK_IN.wAntriebsstatuswort.3
	OR (stEK_IN.wAntriebsstatuswort.8 OR stEK_IN.wAntriebsstatuswort.9 OR stEK_IN.wAntriebsstatuswort.10)
	AND bQ_DRIVE_ENABLE THEN
		stEK_OUT.wSignalsteuerwort.0 := stEK_IN.wSignalstatuswort.10;
	END_IF*)
END_IF


(*##################################################################################*)
(*#### Ausgabe auf zyklische Daten												 ###*)
(*##################################################################################*)

stEK_Out.wSignalsteuerwort.2			:= bInternHoming;
stEK_Out.wSignalsteuerwort.3			:= bABS_REL;
stEK_Out.wSignalsteuerwort.4			:= bIMMEDIATE_CHANGE;
stEK_Out.wSignalsteuerwort.5			:= bRESET;
stEK_Out.wSignalsteuerwort.6			:= bInternJogForward;
stEK_Out.wSignalsteuerwort.7			:= bInternJogBackward ;


stEK_OUT.wMastersteuerwort.13 		:= bInternFrg;


(*####   b.14 is made alwasy on to prevent torque free mode on servo						 ###*)
stEK_OUT.wMastersteuerwort.14 		:= TRUE;


stEK_OUT.wMastersteuerwort.15 		:= bInternHalt;


stEK_OUT.diPositioniergeschwindigkeit 	:= diVEL_CMD;


(*##################################################################################*)
(*#### Einlesen von zyklischen Daten											 ###*)
(*##################################################################################*)

diPOS_ACT 						:= stEK_IN.diLageistwert;
diVEL_ACT 						:= stEK_IN.diIstgeschwindigkeit;
dwDRIVE_DIAGNOSIS 			:= stEK_IN.dwDiagnosenummer;
bSTATUS_MESSAGE 				:= stEK_IN.wAntriebsstatuswort.11;
bWARNING 						:= stEK_IN.wAntriebsstatuswort.12;
bERROR 						:= stEK_IN.wAntriebsstatuswort.13;
bIN_REFERENCE 				:= stEK_IN.wSignalstatuswort.2;
bPOS_OK 						:= stEK_IN.wSignalstatuswort.4;
bIN_STANDSTILL 				:= stEK_IN.wSignalstatuswort.3;
END_FUNCTION_BLOCK

(* POU FB_Indradrive_DCP_using_MUX_8, ST *)
(*#########################################################################################*)
(* General Header *)
(*----------------------------------------------------------------------------------------------------------------------------------------------------------------*)
(* Short description :		      Function Block Drive Controlled positioning using Multiplex Channel“ over      Ethercat *)
(* Version : 					      01VRS                                                                                                                                       *)
(* Name : 					      Upendra Chauhan                                                                                                                    *)
(* Date : 					      2012-02-23                                                                                                                               *)
(* Company : 				      Bosch Rexroth AG                                                                                                                    *)
(* Target : 					      >MPx07VRS                                                                                                                             *)
(* Functional description :		With the help of this function block Indradrive can be used with Drive Contrlled              *)
(*                                                     Positioning mode. The Function block is same as                                                              *)
(*                                                     "FB_DCP_INDRADRIVE_EtherCAT_ST" except the cyclic data transmission.             *)
(*                                                     Here 8 Channel Multiplexer is used for cyclic data read and write. The index used is    *)
(*                                                     predefined as '0'. The required Parameter in AT are configured in Multiplex config list  *)
(*                                                     e.g. S-0-0370, S-0-0490 - S-0-0496 element number '0'                                                   *)
(*                                                     Similarly required MDT parameters are configured in config list S-0-0371, S-0-0500-  *)
(*                                                     S-0-0506 element number '0'                                                                                                 *)
(*----------------------------------------------------------------------------------------------------------------------------------------------------------------*)
(* Handling specials :                                                                                                                                                                      *)
(*----------------------------------------------------------------------------------------------------------------------------------------------------------------*)
(* Additional Header                                                                                                                                                                        *)
(*----------------------------------------------------------------------------------------------------------------------------------------------------------------*)
(* Version : 					 *)
(* Name : 					 *)
(* Date : 						 *)
(* Company : 					 *)
(* *)
(* *)
(* *)
(*-----------------------------------------------------------------------------------------------------------------------------------------------------------------*)
(*##########################################################################################*)
(*##########################################################################################*)
FUNCTION_BLOCK FB_Indradrive_DCP_using_MUX_8
VAR_INPUT
     bDRIVE_ENABLE 					: BOOL; 						(*Antriebstatus Uebergang AB -> AH, Drive Enable state of drive change Ab->AH *)
     bDRIVE_START 					: BOOL; 						(*Antriebstatus Uebergang AH -> AF, Drive Enable state of drive change AH->AF *)
     bHOMING 							: BOOL; 						(*Achse Referenzieren, Homing the axis*)
     bRESET 							: BOOL; 						(*Stoerung quittieren, Reset Error*)
     bJOG_FORWARD 					: BOOL; 						(*Tippen vorwaerts, Jog forward*)
     bJOG_BACKWARD					: BOOL;						(*Tippen rueckwaerts, Jog backward*)
     bNEW_VALUE 						: BOOL; 						(*neuer Sollwert, new value *)
     bABS_REL 						       : BOOL; 						(*Position Absolut = 0 oder Relativ = 1, position = absoluteor relative  *)
     bIMMEDIATE_CHANGE 				: BOOL; 						(*Satzsofortwechsel 1= sofort, immediate block change 1= immediately*)
     diPOS_CMD 						: DINT; 						       (*Soll-Position, Command position*)
     diVEL_CMD 						: DINT; 						       (*Soll-Geschwindigkeit, command velocity*)
     stInputPara                                              : st_Indradrive_DCP_using_MUX_8_input;            (* Input Structure *)
END_VAR
VAR_OUTPUT
     bQ_DRIVE_ENABLE 				: BOOL; 						(*Quittierung DRIVE_ENABLE, acknowledge DRIVE_ENABLE*)
     bQ_MAIN_MODE 					: BOOL; 						(*Quittierung MAIN_MODE, acknowledge MAIN_MODE*)
     bIN_REFERENCE 					: BOOL; 						(*Referenziert, In_Reference*)
     bPOS_OK 							: BOOL; 						(*Sollwert erreicht = 1, target position reached = 1*)
     bNEW_VALUE_POSSIBLE 			: BOOL; 						(*Neuer Sollwert moeglich, NEW_VALUE_POSSIBLE*)
     bSTATUS_MESSAGE 				: BOOL; 						(*STATUS_MESSAGE*)
     bWARNING 						       : BOOL; 						(*WARNING*)
     bERROR 							: BOOL; 						(*ERROR*)
     bIN_STANDSTILL 					: BOOL; 						(*IN_STANDSTILL*)
     dwDRIVE_DIAGNOSIS 				: DWORD; 					       (*DRIVE_DIAGNOSIS*)
     diPOS_ACT 						: DINT; 						       (*Aktuelle Position, actual position*)
     diVEL_ACT 						       : DINT; 						       (*Aktuelle Geschwindigkeit, actual velocity*)
     stOutputPara                                          : st_Indradrive_DCP_using_MUX_8_output;        (* Output Structure *)
END_VAR
VAR
	bInternHalt 						: BOOL; 						(*INTERN_Halt*)
	bInternFrg 						: BOOL; 						(*INTERN_FRG*)
	bInternPosStart 					: BOOL; 						(*INTERN_POS_START*)
	bInternHoming 					: BOOL; 						(*INTERN_HOMING*)
	bInternJogForward 				: BOOL;						(*INTERN_JOG_FORWARD*)
	bInternJogBackward 			: BOOL; 						(*INTERN_JOG_BACKWARD*)
	bNewValueFlanke 				: BOOL; 						(*NEW_VALUE_FLANKE*)
	bNewValueImpulse 				: BOOL; 						(*NEW_VALUE_IMPULSE*)

	wMasterControlWord                   : WORD := 0 ;
	wDriveStatusWord                       : WORD := 0;
	wSignalControlWord                    : WORD := 0 ;
	wSignalStatusWord                     : WORD := 0;
	diPosSetVal                           : DINT := 0;
	diVelSetVal                           : DINT := 0;

	fbMuxIndradrive                             : FB_Indradrive_MUX_8 ;

END_VAR
(*##################################################################################*)
(*#### Read Cyclic Data from Drive                                                                                                                      ###*)
(*##################################################################################*)
(* Convert Parameter specific datatypes to DWORD *)
wDriveStatusWord                   := DWORD_TO_WORD (stInputPara.wDriveStatusWord);
wSignalStatusWord                  := DWORD_TO_WORD (fbMuxIndradrive.dwValue_READ_2);
diVEL_ACT                               := DWORD_TO_DINT (fbMuxIndradrive.dwValue_READ_3);
diPOS_ACT                              := DWORD_TO_DINT (fbMuxIndradrive.dwValue_READ_4);
dwDRIVE_DIAGNOSIS           := fbMuxIndradrive.dwValue_READ_5;

bSTATUS_MESSAGE            := wDriveStatusWord.11;
bWARNING                               := wDriveStatusWord.12;
bERROR                                   := wDriveStatusWord.13;
bIN_REFERENCE                  := wSignalStatusWord.2;
bPOS_OK                                := wSignalStatusWord.4;
bIN_STANDSTILL                   := wSignalStatusWord.3;

(*##################################################################################*)
(*####  Preparing Status values                                                                                                                             ###*)
(*##################################################################################*)
(* Drive in AF? *)
bQ_DRIVE_ENABLE			:= wDriveStatusWord.14 AND wDriveStatusWord.15;

(* Drive enabled (in AF) + Drive Follows Cmd + Primary OpMode active *)
bQ_MAIN_MODE 				:= wDriveStatusWord.3
									AND bQ_DRIVE_ENABLE
									AND NOT wDriveStatusWord.8
									AND NOT wDriveStatusWord.9
									AND NOT wDriveStatusWord.10;

bNEW_VALUE_POSSIBLE		:=   NOT ( wSignalControlWord.0 XOR wSignalStatusWord.10) AND  (* both are zero or both are one *)
									bQ_MAIN_MODE AND                                                                        (* Drive in AF *)
									bInternPosStart;                                                                                     (* Positioning is already active *)

(*##################################################################################*)
(*####  Preparing Command values                                                                                                                      ###*)
(*##################################################################################*)

bInternHoming 					:= bInternFrg AND NOT bInternPosStart AND NOT bJOG_FORWARD
									AND NOT bJOG_BACKWARD AND bHOMING;

bInternJogForward 				:= bInternFrg AND NOT bInternPosStart AND bJOG_FORWARD
									AND NOT bJOG_BACKWARD AND NOT bHOMING;

bInternJogBackward 			:= bInternFrg AND NOT bInternPosStart AND NOT bJOG_FORWARD
									AND bJOG_BACKWARD AND NOT bHOMING;

bInternPosStart					:= bInternFrg AND NOT bJOG_FORWARD
									AND NOT bJOG_BACKWARD AND NOT bHOMING;

bInternHalt						:= bDRIVE_ENABLE;

bInternFrg 						:= bInternHalt AND bQ_DRIVE_ENABLE AND bDRIVE_START;

(*##################################################################################*)
(*####  Bildung Togglebit für Sollwertübernahme 								 ###*)
(*##################################################################################*)
bNewValueImpulse				:= bNEW_VALUE AND NOT bNewValueFlanke;
bNewValueFlanke				:= bNEW_VALUE;

IF (bNEW_VALUE_POSSIBLE OR bIMMEDIATE_CHANGE) AND bInternPosStart AND bNewValueImpulse THEN
	(* assign Position Command value *)
	diPosSetVal := diPOS_CMD;

	(* toggle bit 0 of wSignalControlWord to accept new commanded values *)
	IF   (wSignalControlWord.0 XOR wSignalStatusWord.10 ) AND (* when both are not same ( 1 , 0 or 0 , 1)*)
		bIMMEDIATE_CHANGE
	THEN
		(* accept immediatly *)
		wSignalControlWord.0 := wSignalStatusWord.10;
	ELSE (* if both are same ( 0 ,0) or ( 1, 1) or Immediate Change is requested *)
		(* accept at next command *)
		wSignalControlWord.0 := NOT wSignalStatusWord.10;
	END_IF

(*Verhinderung F2050 -->nicht nötig Anwenderfehler sollen zu Antriebsfehlern führen*)
(*ELSE
	IF wDriveStatusWord.3
	OR (wDriveStatusWord.8 OR wDriveStatusWord.9 OR wDriveStatusWord.10)
	AND bQ_DRIVE_ENABLE THEN
		wSignalControlWord.0 := wSignalStatusWord.10;
	END_IF*)
END_IF
(* assign Velocity for positioning, value will only be taken over when bit 0 of wSignalControlWord is toggled *)
diVelSetVal 	:= diVEL_CMD;

(* set Master Control Word for Drive *)
wMasterControlWord.13		:= bInternFrg;
wMasterControlWord.14 		:= bInternHalt;
wMasterControlWord.15 		:= bInternHalt;

(* set Signal Control Word for Drive *)
wSignalControlWord.2			:= bInternHoming;
wSignalControlWord.3			:= bABS_REL;
wSignalControlWord.4			:= bIMMEDIATE_CHANGE;
wSignalControlWord.5			:= bRESET;
wSignalControlWord.6			:= bInternJogForward;
wSignalControlWord.7			:= bInternJogBackward ;


(*##################################################################################*)
(*#### Ausgabe auf zyklische Daten												 ###*)
(*##################################################################################*)
stOutputPara.wMasterControlWord := wMasterControlWord;
(* Convert DWORD value to corresponding data type as per the Parameter DataType *)
fbMuxIndradrive.dwValue_WRITE_2 := WORD_TO_DWORD ( wSignalControlWord);
fbMuxIndradrive.dwValue_WRITE_3 := DINT_TO_DWORD  ( diVelSetVal);
fbMuxIndradrive.dwValue_WRITE_4 := DINT_TO_DWORD  ( diPosSetVal);

(*###############################################################################*)
(*####  Call Multiplex Function block and get element number '0' Read and Written Cyclically                      *)
(*###############################################################################*)
fbMuxIndradrive(
	uiINDEX_WRITE                          := OP_MODE_DCP ,
	uiLIST_INDEX_WRITE                := LIST_INDEX_0,
	dwValue_WRITE_1                     :=  ,       (* S-0-0000 - Reserve *)
	dwValue_WRITE_2                     :=  ,       (* S-0-0145 - Signal control word *)
	dwValue_WRITE_3                     :=  ,       (* S-0-0259 - Positioning Velocity*)
	dwValue_WRITE_4                     :=  ,       (* S-0-0282 - Position Command Value *)
	dwValue_WRITE_5                     :=  ,       (* S-0-0000 - Reserve *)
	dwValue_WRITE_6                     :=  ,       (* S-0-0000 - Reserve *)
	dwValue_WRITE_7                     :=  ,       (* S-0-0000 - Reserve *)
	dwValue_WRITE_8                     :=  ,       (* S-0-0000 - Reserve *)
	uiINDEX_READ                           := OP_MODE_DCP,
	uiLIST_INDEX_READ                 := LIST_INDEX_0 ,
	stEK_IN                                         := stInputPara.stMUX_in ,
	uiINDEX_WRITE_ACKNOWLEDGE=> ,
	uiLIST_INDEX_WRITE_ACKNOWLEDGE=> ,
	uiINDEX_READ_ACKNOWLEDGE=> ,
	uiLIST_INDEX_READ_ACKNOWLEDGE=> ,
	dwValue_READ_1                      => ,           (* S-0-0000 - Reserve *)
	dwValue_READ_2                      => ,           (* S-0-0144 - Signal Status word *)
	dwValue_READ_3                      => ,           (* S-0-0047 - Velocity feedback value *)
	dwValue_READ_4                      => ,           (* S-0-0051 - Postion feedback value *)
	dwValue_READ_5                      => ,           (* S-0-0390 - Drive Diagnostic word *)
	dwValue_READ_6                      => ,           (* S-0-0000 - Reserve *)
	dwValue_READ_7                      => ,           (* S-0-0000 - Reserve *)
	dwValue_READ_8                      => ,           (* S-0-0000 - Reserve *)
	stEK_OUT                                    => stOutputPara.stMUX_out);
END_FUNCTION_BLOCK

(* POU FB_Indradrive_MUX_8, IL *)
FUNCTION_BLOCK FB_Indradrive_MUX_8

VAR_INPUT
	uiINDEX_WRITE 			: UINT:= 0; (*S-0-0368, Bit 0-5 Adressing for Data Container A MDT Select*)
    	uiLIST_INDEX_WRITE 		: UINT:= 0; (*S-0-0362 List index, MDT Data Container A*)
    	dwValue_WRITE_1 		: DWORD:= 0; (*S-0-0360 MDT Data Container A*)
    	dwValue_WRITE_2 		: DWORD := 0; (*S-0-0450 MDT Data Container A*)
    	dwValue_WRITE_3 		: DWORD := 0; (*S-0-0451 MDT Data Container A*)
    	dwValue_WRITE_4 		: DWORD := 0; (*S-0-0452 MDT Data Container A*)
    	dwValue_WRITE_5 		: DWORD := 0; (*S-0-0453 MDT Data Container A*)
    	dwValue_WRITE_6 		: DWORD := 0; (*S-0-0454 MDT Data Container A*)
    	dwValue_WRITE_7 		: DWORD := 0; (*S-0-0455 MDT Data Container A*)
    	dwValue_WRITE_8 		: DWORD := 0; (*S-0-0456 MDT Data Container A*)
   	uiINDEX_READ 			: UINT:= 0; (*S-0-0368 Bit 8-13 Adresssing for data container A AT Acknowledge*)
   	uiLIST_INDEX_READ 		: UINT:= 0; (*S-0-0366 List index, AT Data Container A*)
	stEK_IN 				: st_Indradrive_MUX_8_input;
END_VAR

VAR_OUTPUT
	uiINDEX_WRITE_ACKNOWLEDGE 			: UINT:= 0; (*S-0-0368, Bit 0-5 Adressing for Data Container A MDT Select*)
  	uiLIST_INDEX_WRITE_ACKNOWLEDGE 		: UINT:= 0; (*S-0-0362 List index, MDT Data Container A*)
   	uiINDEX_READ_ACKNOWLEDGE 			: UINT:= 0; (*S-0-0368 Bit 8-13 Adresssing for data container A AT Acknowledge*)
	uiLIST_INDEX_READ_ACKNOWLEDGE		: UINT:= 0; (*S-0-0366 List index, AT Data Container A*)
	dwValue_READ_1						: DWORD := 0; (*S-0-0364 AT Data Container A*)
	dwValue_READ_2						: DWORD := 0; (*S-0-0480 AT Data Container A*)
	dwValue_READ_3						: DWORD := 0; (*S-0-0481 AT Data Container A*)
	dwValue_READ_4						: DWORD := 0; (*S-0-0482 AT Data Container A*)
	dwValue_READ_5						: DWORD := 0; (*S-0-0483 AT Data Container A*)
	dwValue_READ_6						: DWORD := 0; (*S-0-0484 AT Data Container A*)
	dwValue_READ_7						: DWORD := 0; (*S-0-0485 AT Data Container A*)
	dwValue_READ_8						: DWORD := 0; (*S-0-0486 AT Data Container A*)
	stEK_OUT 			: st_Indradrive_MUX_8_output;
END_VAR

VAR_IN_OUT
END_VAR

VAR
	wInternIndexWrite		: WORD;
	wInternIndexRead		: WORD;
END_VAR
	(*Schreiben über den Multiplexkanal / Write via multiplex channel*)
	
	(*Auswahl eines in S-0-0370 (Konfigurationsliste MDT-Datencontainer) konfigurierten Parameters, der beschrieben werden soll*)
	(*Select a parameter from S-0-0370 (Configuration list for the MDT-data container), which should be written*)
	
	LD		uiINDEX_WRITE
	UINT_TO_WORD
	ST		wInternIndexWrite
	
	LD		wInternIndexWrite.0
	ST		stEK_OUT.uiIndexAdressing.0
	
	LD		wInternIndexWrite.1
	ST		stEK_OUT.uiIndexAdressing.1
	
	LD		wInternIndexWrite.2
	ST		stEK_OUT.uiIndexAdressing.2
	
	LD		wInternIndexWrite.3
	ST		stEK_OUT.uiIndexAdressing.3
	
	LD		wInternIndexWrite.4
	ST		stEK_OUT.uiIndexAdressing.4
	
	LD		wInternIndexWrite.5
	ST		stEK_OUT.uiIndexAdressing.5
	
	(*Auswahl eines Elements bei Listenparamtern  (S-0-0362*)
	(*Select a single element from the list paramter (S-0-0362*)
	
	LD		uiLIST_INDEX_WRITE
	ST		stEK_OUT.uiListIndexWrite
	
	(*Beschreiben des MDT-Datencontainers A Wert 1 (S-0-0360) mit einem Wert*)
	(* Write a value in the MDT-data-Container A value 1 (S-0-0360*)
	LD		dwValue_WRITE_1
	ST		stEK_OUT.dwWriteValue1
	
	(*Beschreiben des MDT-Datencontainers A Wert 2 (S-0-0450) mit einem Wert*)
	(* Write a value in the MDT-data-Container A value 2 (S-0-0450*)
	LD		dwValue_WRITE_2
	ST		stEK_OUT.dwWriteValue2

	(*Beschreiben des MDT-Datencontainers A Wert 3 (S-0-0451) mit einem Wert*)
	(* Write a value in the MDT-data-Container A value 3 (S-0-0451*)
	LD		dwValue_WRITE_3
	ST		stEK_OUT.dwWriteValue3

	(*Beschreiben des MDT-Datencontainers A Wert 4 (S-0-0452) mit einem Wert*)
	(* Write a value in the MDT-data-Container A value 4 (S-0-0452*)
	LD		dwValue_WRITE_4
	ST		stEK_OUT.dwWriteValue4

	(*Beschreiben des MDT-Datencontainers A Wert 5 (S-0-0453) mit einem Wert*)
	(* Write a value in the MDT-data-Container A value 5 (S-0-0453*)
	LD		dwValue_WRITE_5
	ST		stEK_OUT.dwWriteValue5

	(*Beschreiben des MDT-Datencontainers A Wert 6 (S-0-0454) mit einem Wert*)
	(* Write a value in the MDT-data-Container A value 6 (S-0-0454*)
	LD		dwValue_WRITE_6
	ST		stEK_OUT.dwWriteValue6

	(*Beschreiben des MDT-Datencontainers A Wert 7 (S-0-0455) mit einem Wert*)
	(* Write a value in the MDT-data-Container A value 7 (S-0-0455*)
	LD		dwValue_WRITE_7
	ST		stEK_OUT.dwWriteValue7

	(*Beschreiben des MDT-Datencontainers A Wert 8 (S-0-0456) mit einem Wert*)
	(* Write a value in the MDT-data-Container A value 8 (S-0-0456*)
	LD		dwValue_WRITE_8
	ST		stEK_OUT.dwWriteValue8

	(*Anzeigen der Rückmeldung  (S-0-0368, Bit 0-5) "INDEX_WRITE_ACKNOWLEDGE"*)
	(*Show the acknowledge (S-0-0368, Bit 0-5)  "INDEX_WRITE_ACKNOWLEDGE"*)
	
	LD		stEK_IN.uiIndexAdressing.0
	ST		uiINDEX_WRITE_ACKNOWLEDGE.0
	
	LD		stEK_IN.uiIndexAdressing.1
	ST		uiINDEX_WRITE_ACKNOWLEDGE.1
	
	LD		stEK_IN.uiIndexAdressing.2
	ST		uiINDEX_WRITE_ACKNOWLEDGE.2
	
	LD		stEK_IN.uiIndexAdressing.3
	ST		uiINDEX_WRITE_ACKNOWLEDGE.3
	
	LD		stEK_IN.uiIndexAdressing.4
	ST		uiINDEX_WRITE_ACKNOWLEDGE.4
	
	LD		stEK_IN.uiIndexAdressing.5
	ST		uiINDEX_WRITE_ACKNOWLEDGE.5
	
	
	(*Anzeigen der Rückmeldung (S-0-0362) "LIST _INDEX_WRITE_ACKNOWLEDGE"*)
	(*Show the acknowledge (S-0-0362) "LIST _INDEX_WRITET_ACKNOWLEDGE*)
	
	LD		stEK_IN.uiListIndexWrite
	ST		uiLIST_INDEX_WRITE_ACKNOWLEDGE
	
	
	(*Lesen über den Multiplexkanal / Read via multiplex channel*)
	
	(*Auswahl eines in S-0-0371 (Konfigurationsliste AT-Datencontainer) konfigurierten Parameters, der gelesen werden soll*)
	(*Select a parameter from S-0-0371 (Configuration list for the AT-data container), which should be read*)
	
	LD		uiINDEX_READ
	UINT_TO_WORD
	ST		wInternIndexRead
	
	LD		wInternIndexRead.0
	ST		stEK_OUT.uiIndexAdressing.8
	
	LD		wInternIndexRead.1
	ST		stEK_OUT.uiIndexAdressing.9
	
	LD		wInternIndexRead.2
	ST		stEK_OUT.uiIndexAdressing.10
	
	LD		wInternIndexRead. 3
	ST		stEK_OUT.uiIndexAdressing.11
	
	LD		wInternIndexRead.4
	ST		stEK_OUT.uiIndexAdressing.12
	
	LD		wInternIndexRead.5
	ST		stEK_OUT.uiIndexAdressing.13

	
	(*Auswahl eines Elements bei einem Listenparameter (S-0-0366*)
	(*Select a single element from the list parameter (S-0-0366 *)
	
	LD		uiLIST_INDEX_READ
	ST		stEK_OUT.uiListIndexRead
	
	(*Anzeigen der Rückmeldung (S-0-0368, Bit 8-13) "INDEX_READ_ACKNOWLEDGE"*)
	(*Show the acknowledge (S-0-0368, Bit 8-13)  "INDEX_READ_ACKNOWLEDGE"*)
	
	LD		stEK_IN.uiIndexAdressing.8
	ST		uiINDEX_READ_ACKNOWLEDGE.0
	
	LD		stEK_IN.uiIndexAdressing.9
	ST		uiINDEX_READ_ACKNOWLEDGE.1
	
	LD		stEK_IN.uiIndexAdressing.10
	ST		uiINDEX_READ_ACKNOWLEDGE.2
	
	LD		stEK_IN.uiIndexAdressing.11
	ST		uiINDEX_READ_ACKNOWLEDGE.3
	
	LD		stEK_IN.uiIndexAdressing.12
	ST		uiINDEX_READ_ACKNOWLEDGE.4
	
	LD		stEK_IN.uiIndexAdressing.13
	ST		uiINDEX_READ_ACKNOWLEDGE.5
	
	(*Anzeigen der Rückmeldung (S-0-0366) "LIST_INDEX_READ_ACKNOWLEDGE"*)
	(*Show the acknowledge (S-0-0366) "LIST_INDEX_READ_ACKNOWLEDGE*)
	
	LD		stEK_IN.uiListIndexRead
	ST		uiLIST_INDEX_READ_ACKNOWLEDGE
	
	(*Anzeigen des Wertes des zu lesenden Parameters (S-0-0364) "VALUE_READ_1"*)
	(*Show the value which was read from a parameter (S-0-0364)  "VALUE_READ_1"*)
	LD		stEK_IN.dwReadValue1
	ST		dwValue_READ_1
	
	(*Anzeigen des Wertes des zu lesenden Parameters (S-0-0480) "VALUE_READ_2"*)
	(*Show the value which was read from a parameter (S-0-0480)  "VALUE_READ_2"*)
	LD		stEK_IN.dwReadValue2
	ST		dwValue_READ_2

	(*Anzeigen des Wertes des zu lesenden Parameters (S-0-0481) "VALUE_READ_3"*)
	(*Show the value which was read from a parameter (S-0-0481)  "VALUE_READ_3"*)
	LD		stEK_IN.dwReadValue3
	ST		dwValue_READ_3

	(*Anzeigen des Wertes des zu lesenden Parameters (S-0-0482) "VALUE_READ_4"*)
	(*Show the value which was read from a parameter (S-0-0482)  "VALUE_READ_4"*)
	LD		stEK_IN.dwReadValue4
	ST		dwValue_READ_4

	(*Anzeigen des Wertes des zu lesenden Parameters (S-0-0483) "VALUE_READ_5"*)
	(*Show the value which was read from a parameter (S-0-0483)  "VALUE_READ_5"*)
	LD		stEK_IN.dwReadValue5
	ST		dwValue_READ_5

	(*Anzeigen des Wertes des zu lesenden Parameters (S-0-0484) "VALUE_READ_6"*)
	(*Show the value which was read from a parameter (S-0-0484)  "VALUE_READ_6"*)
	LD		stEK_IN.dwReadValue6
	ST		dwValue_READ_6

	(*Anzeigen des Wertes des zu lesenden Parameters (S-0-0485) "VALUE_READ_7"*)
	(*Show the value which was read from a parameter (S-0-0485)  "VALUE_READ_7"*)
	LD		stEK_IN.dwReadValue7
	ST		dwValue_READ_7

	(*Anzeigen des Wertes des zu lesenden Parameters (S-0-0486) "VALUE_READ_8"*)
	(*Show the value which was read from a parameter (S-0-0486)  "VALUE_READ_8"*)
	LD		stEK_IN.dwReadValue8
	ST		dwValue_READ_8
END_FUNCTION_BLOCK

(* POU FB_Indradrive_MUX_1, IL *)
FUNCTION_BLOCK FB_Indradrive_MUX_1

VAR_INPUT
	uiINDEX_WRITE 			: UINT:= 0; (*S-0-0368, Bit 0-5 Adressing for Data Container A MDT Select*)
    	uiLIST_INDEX_WRITE 		: UINT:= 0; (*S-0-0362 List index, MDT Data Container A*)
    	diVALUE_WRITE_1 		: DINT:= 0; (*S-0-0360 MDT Data Container A*)
   	uiINDEX_READ 			: UINT:= 0; (*S-0-0368 Bit 8-13 Adresssing for data container A AT Acknowledge*)
   	uiLIST_INDEX_READ 		: UINT:= 0; (*S-0-0366 List index, AT Data Container A*)
	stEK_IN 				: st_Indradrive_MUX_1_input;
END_VAR

VAR_OUTPUT
	uiINDEX_WRITE_ACKNOWLEDGE 			: UINT:= 0; (*S-0-0368, Bit 0-5 Adressing for Data Container A MDT Select*)
  	uiLIST_INDEX_WRITE_ACKNOWLEDGE 		: UINT:= 0; (*S-0-0362 List index, MDT Data Container A*)
   	uiINDEX_READ_ACKNOWLEDGE 			: UINT:= 0; (*S-0-0368 Bit 8-13 Adresssing for data container A AT Acknowledge*)
	uiLIST_INDEX_READ_ACKNOWLEDGE		: UINT:= 0; (*S-0-0366 List index, AT Data Container A*)
	diVALUE_READ_1						: DINT:= 0; (*S-0-0364 AT Data Container A*)
	stEK_OUT 			: st_Indradrive_MUX_1_output;
END_VAR

VAR_IN_OUT
END_VAR

VAR
	wInternIndexWrite		: WORD;
	wInternIndexRead		: WORD;
END_VAR
	(*Schreiben über den Multiplexkanal / Write via multiplex channel*)
	
	(*Auswahl eines in S-0-0370 (Konfigurationsliste MDT-Datencontainer) konfigurierten Parameters, der beschrieben werden soll*)
	(*Select a parameter from S-0-0370 (Configuration list for the MDT-data container), which should be written*)
	
	LD		uiINDEX_WRITE
	UINT_TO_WORD
	ST		wInternIndexWrite
	
	LD		wInternIndexWrite.0
	ST		stEK_OUT.uiIndexAdressing.0
	
	LD		wInternIndexWrite.1
	ST		stEK_OUT.uiIndexAdressing.1
	
	LD		wInternIndexWrite.2
	ST		stEK_OUT.uiIndexAdressing.2
	
	LD		wInternIndexWrite.3
	ST		stEK_OUT.uiIndexAdressing.3
	
	LD		wInternIndexWrite.4
	ST		stEK_OUT.uiIndexAdressing.4
	
	LD		wInternIndexWrite.5
	ST		stEK_OUT.uiIndexAdressing.5
	
	(*Auswahl eines Elements bei Listenparamtern  (S-0-0362*)
	(*Select a single element from the list paramter (S-0-0362*)
	
	LD		uiLIST_INDEX_WRITE
	ST		stEK_OUT.uiListIndexWrite
	
	(*Beschreiben des MDT-Datencontainers A Wert 1 (S-0-0360) mit einem Wert*)
	(* Write a value in the MDT-data-Container A value 1 (S-0-0360*)
	
	LD		diVALUE_WRITE_1
	ST		stEK_OUT.diWriteValue1
	
	
	(*Anzeigen der Rückmeldung  (S-0-0368, Bit 0-5) "INDEX_WRITE_ACKNOWLEDGE"*)
	(*Show the acknowledge (S-0-0368, Bit 0-5)  "INDEX_WRITE_ACKNOWLEDGE"*)
	
	LD		stEK_IN.uiIndexAdressing.0
	ST		uiINDEX_WRITE_ACKNOWLEDGE.0
	
	LD		stEK_IN.uiIndexAdressing.1
	ST		uiINDEX_WRITE_ACKNOWLEDGE.1
	
	LD		stEK_IN.uiIndexAdressing.2
	ST		uiINDEX_WRITE_ACKNOWLEDGE.2
	
	LD		stEK_IN.uiIndexAdressing.3
	ST		uiINDEX_WRITE_ACKNOWLEDGE.3
	
	LD		stEK_IN.uiIndexAdressing.4
	ST		uiINDEX_WRITE_ACKNOWLEDGE.4
	
	LD		stEK_IN.uiIndexAdressing.5
	ST		uiINDEX_WRITE_ACKNOWLEDGE.5
	
	
	(*Anzeigen der Rückmeldung (S-0-0362) "LIST _INDEX_WRITE_ACKNOWLEDGE"*)
	(*Show the acknowledge (S-0-0362) "LIST _INDEX_WRITET_ACKNOWLEDGE*)
	
	LD		stEK_IN.uiListIndexWrite
	ST		uiLIST_INDEX_WRITE_ACKNOWLEDGE
	
	
    (*Lesen über den Multiplexkanal / Read via multiplex channel*)
	
    (*Auswahl eines in S-0-0371 (Konfigurationsliste AT-Datencontainer) konfigurierten Parameters, der gelesen werden soll*)
	(*Select a parameter from S-0-0371 (Configuration list for the AT-data container), which should be read*)
	
	LD		uiINDEX_READ
	UINT_TO_WORD
	ST		wInternIndexRead
	
	LD		wInternIndexRead.0
	ST		stEK_OUT.uiIndexAdressing.8
	
	LD		wInternIndexRead.1
	ST		stEK_OUT.uiIndexAdressing.9
	
	LD		wInternIndexRead.2
	ST		stEK_OUT.uiIndexAdressing.10
	
	LD		wInternIndexRead. 3
	ST		stEK_OUT.uiIndexAdressing.11
	
	LD		wInternIndexRead.4
	ST		stEK_OUT.uiIndexAdressing.12
	
	LD		wInternIndexRead.5
	ST		stEK_OUT.uiIndexAdressing.13

	
	(*Auswahl eines Elements bei einem Listenparameter (S-0-0366*)
	(*Select a single element from the list parameter (S-0-0366 *)
	
	LD		uiLIST_INDEX_READ
	ST		stEK_OUT.uiListIndexRead
	
	(*Anzeigen der Rückmeldung (S-0-0368, Bit 8-13) "INDEX_READ_ACKNOWLEDGE"*)
	(*Show the acknowledge (S-0-0368, Bit 8-13)  "INDEX_READ_ACKNOWLEDGE"*)
	
	LD		stEK_IN.uiIndexAdressing.8
	ST		uiINDEX_READ_ACKNOWLEDGE.0
	
	LD		stEK_IN.uiIndexAdressing.9
	ST		uiINDEX_READ_ACKNOWLEDGE.1
	
	LD		stEK_IN.uiIndexAdressing.10
	ST		uiINDEX_READ_ACKNOWLEDGE.2
	
	LD		stEK_IN.uiIndexAdressing.11
	ST		uiINDEX_READ_ACKNOWLEDGE.3
	
	LD		stEK_IN.uiIndexAdressing.12
	ST		uiINDEX_READ_ACKNOWLEDGE.4
	
	LD		stEK_IN.uiIndexAdressing.13
	ST		uiINDEX_READ_ACKNOWLEDGE.5
	
	(*Anzeigen der Rückmeldung (S-0-0366) "LIST_INDEX_READ_ACKNOWLEDGE"*)
	(*Show the acknowledge (S-0-0366) "LIST_INDEX_READ_ACKNOWLEDGE*)
	
	LD		stEK_IN.uiListIndexRead
	ST		uiLIST_INDEX_READ_ACKNOWLEDGE
	
	(*Anzeigen des Wertes des zu lesenden Parameters (S-0-0364) "VALUE_READ_1"*)
	(*Show the value which was read from a parameter (S-0-0364)  "VALUE_READ_1"*)
	
	LD		stEK_IN.diReadValue1
	ST		diVALUE_READ_1
END_FUNCTION_BLOCK

(* POU FB_Process_Control, ST *)
(*#################################################################################################*)
(* General Header                                                                                                                                                                                             *)
(*------------------------------------------------------------------------------------------------------------------------------------------------------------------------------*)
(* Short description :               Function Block "FB_Process_control" controls Process values using MLD program                           *)
(* Version :                                 01VRS                                                                                                                                                           *)
(* Name :                                    Upendra Chauhan                                                                                                                                        *)
(* Date :                                       2012-08-20                                                                                                                                                  *)
(* Company :                             Bosch Rexroth AG                                                                                                                                         *)
(* Target :´                                  >MPx07VRS                                                                                                                                                  *)
(* Functional description :      The "FB_Process_Control" FUNCTION block provides a user interface for the                      *)
(*                                                     Process control FUNCTION block available in the Indradrive using MLD. In addition          *)
(*                                                     to the interface FOR Pressure control, this FB also gives a possibility OF using                     *)
(*                                                     Flow rate control instead OF the Pressure control. This FB uses Multiplex channel               *)
(*                                                     (8 Channels) FOR cyclic data communication between Control AND Indradrive                     *)
(*--------------------------------------------------------------------------------------------------------------------------------------------------------------------------*)
(* Handling specials :                                                                                                                                                                                           *)
(*--------------------------------------------------------------------------------------------------------------------------------------------------------------------------*)
(* Additional Header                                                                                                                                                                                             *)
(*--------------------------------------------------------------------------------------------------------------------------------------------------------------------------*)
(* Version : 1.0	                                                                                                                                                                                                *)
(* Name : urc2kor ( DC-IA/EDY )                                                                                                                                                                       *)
(* Date : 08,05,2012                                                                                                                                                                                                *)
(* Company : Bosch Rexroth                                                                                                                                                                              *)
(*--------------------------------------------------------------------------------------------------------------------------------------------------------------------------*)
(* Version : 1.1	                                                                                                                                                                                           *)
(* Name : urc2kor ( DC-IA/EDY )                                                                                                                                                               *)
(* Date : 29.10.2012                                                                                                                                                                                   *)
(* Company : Bosch Rexroth                                                                                                                                                                      *)
(* Drive Halt Bit activated with DriveStart Input. Without this it is not possible to Activate AF mode at Drive                                   *)
(*--------------------------------------------------------------------------------------------------------------------------------------------------------------------------*)
(* Version : 1.1	                                                                                                                                                                                           *)
(* Name : urc2kor ( DC-IA/EDY )                                                                                                                                                               *)
(* Date : 29.10.2012                                                                                                                                                                                   *)
(* Company : Bosch Rexroth                                                                                                                                                                      *)
(* Drive Halt Bit activated with DriveStart Input. Without this it is not possible to Activate AF mode at Drive                                   *)
(*--------------------------------------------------------------------------------------------------------------------------------------------------------------------------*)
(* Version : 1.2	                                                                                                                                                                                           *)
(* Name : urc2kor ( DC-IA/EDY )                                                                                                                                                               *)
(* Date : 11.12.2012                                                                                                                                                                                   *)
(* Company : Bosch Rexroth                                                                                                                                                                      *)
(* Drive Halt acknoledgement is configured in SignalStatusWord Bit-5. Bit 3-4 was wrong, corrected the same.                          *)
(* Process control was deactivated when the DriveStart or DriveEnable is removed.                                                                        *)
(*------------------------------------------------------------------------------------------------------------------------------------------------------------------------*)
(* Version : 1.3	                                                                                                                                                                                              *)
(* Name : urc2kor ( DC-IA/EDY )                                                                                                                                                                     *)
(*Date: 18.02.2013                                                                                                                                                                                                *)
(* Company : Bosch Rexroth                                                                                                                                                                            *)
(* "Process Control FB" updated with possibility OF using Pressure Value AND Flowrate values in Percentage             *)
(* Selection OF the Parameter Set is now possible with Input field by Changing bit 7,8 of P-1390                                            *)
(* New Input 'InjectionPhaseActive' added and passed on to bit 3 of P-1390                                                                                 *)
(* Added new cyclic input 'wAxisControllerMessage' (P-0-0555). Signal Status word setting made same as MLC/MLD *)
(* Added new cyclic output 'diVelocityLimitPos' (P-0-1377). Limit value calculated while in Pressure control and in         *)
(* case of Flow control defaul value pased on to the limit.                                                                                                                      *)
(*------------------------------------------------------------------------------------------------------------------------------------------------------------------------*)
(* Version : 1.4	                                                                                                                                                                                              *)
(* Name : raa2bmh ( DC-IA/EDY )                                                                                                                                                                   *)
(*Date: 20.08.2014                                                                                                                                                                                                *)
(* Company : Bosch Rexroth                                                                                                                                                                            *)
(* "Process Control FB" updated with drive enable ad drive halt change in bits							             *)
(* Volume multiplication factor is changed from 10000 to 10.											             *)
(*------------------------------------------------------------------------------------------------------------------------------------------------------------------------*)
(*#################################################################################################*)
(*#################################################################################################*)
FUNCTION_BLOCK FB_Process_Control
VAR_INPUT
	DriveEnable : BOOL;
	DriveStart : BOOL;
	ResetDriveError : BOOL;
	PumpOn : BOOL;
	InjectionPhaseActive : BOOL;
	OperatingMode : INT;
	PressureCmdValue : REAL;
	FlowrateCmdValue : REAL;
	VolumePump01 : REAL;
	VolumePump02 : REAL;
	PressureUnit : UINT;
	FlowrateUnit : UINT;
	NominalPressureValue : REAL;(*REAL*)
	NominalFlowrateValue : REAL;(*REAL*)
	ParameterSetNo : UINT;
	stInputPara : st_Indradrive_ProcessControl_input;
END_VAR
VAR_OUTPUT
	DriveState : INT;
	InStandstill : BOOL;
	CommandValueReached : BOOL;
	Pump01On : BOOL;
	Pump02On: BOOL;
	VelocityHighLimitActive: BOOL;
	VelocityLowLevelWarning: BOOL;
	TorqueHighLimitActive : BOOL;
	ProcessOutputHLActive : BOOL;
	ProcessOutputLLActive:BOOL;
	ProcessControlError : BOOL;
	DriveWarning: BOOL;
	DriveError: BOOL;
	PressureActValue : REAL;
	FlowrateActValue: REAL;
	DriveDiagnosis : DWORD;
	ActiveParameterSetNo : UINT;
	stOutputPara : st_Indradrive_ProcessControl_output;
END_VAR
VAR
	wMasterControlWord                   : WORD := 0 ;
	wDriveStatusWord                       : WORD := 0;
	wSignalControlWord                    : WORD := 0 ;
	wSignalStatusWord                     : WORD := 0;

	diVelocityAct: DINT := 0;
	rVelocityAct: REAL := 0;
	wMLDStatusWord: WORD;
	bMLDPump2OnCmd: BOOL := FALSE;
	bMLDRunning: BOOL := FALSE;
	bPressureControlActive: BOOL := FALSE;
	bPressureCmdValReached: BOOL := FALSE;
	bOpModeAck_bit0: BOOL := FALSE;
	bOpModeAck_bit1: BOOL := FALSE;
	bDriveHalt: BOOL := FALSE;
	bModePMActive: BOOL := FALSE;
	bVelCmdValReached: BOOL := FALSE;
	bOpModeAck_bit2: BOOL := FALSE;
	bDriveMessageClass3: BOOL := FALSE;
	DriveMode: WORD := 0;
	dwTotalVolume: REAL := 0;
	diVelocityCmd: DINT := 0;
	diPressureCmd: DINT := 0;
	wMLDControlWord: WORD := 0;
	FlowrateActValueInternal: REAL;
	PressureCmdValueInternal: REAL;
	PressureActValueInternal: REAL;
	FlowrateCmdValueInternal: REAL;
	diVelocityLimitPos: DINT;
	wAxisMessages: WORD;
	uiParameterSetNoInternal:UINT;
	uiActiveParameterSetNoInternal: UINT;
END_VAR

VAR CONSTANT
	PERCENTAGE_BASE : DINT := 100;
	DEC_POINT_ADJUSTMENT : DINT := 100;
	DEFAULT_N_POSITIVE_LIMIT : REAL := 3000;
	CONV_FACTOR_DWORDTOREAL:REAL:=10000;
	CONV_FACTOR_REALTODWORD:REAL:=10000;
	CONV_FACTOR_VOLUME:REAL:=10;
END_VAR
(* Read Actual values from Drive *)
(* Convert Parameter specific datatypes to DWORD *)
wDriveStatusWord                   := DWORD_TO_WORD (stInputPara.wDriveStatusWord);
wSignalStatusWord                  := DWORD_TO_WORD (stInputPara.wSignalStatusWord);
wMLDStatusWord                    := DWORD_TO_WORD (stInputPara.wProcessControlStatusWord);
wAxisMessages                      := DWORD_TO_WORD (stInputPara.wAxisControllerMessage);

diVelocityAct                             :=stInputPara.diVelocityAct;
rVelocityAct                               := DINT_TO_REAL(diVelocityAct) / CONV_FACTOR_DWORDTOREAL;
PressureActValueInternal     := DWORD_TO_REAL(stInputPara.diPressureAct) /  CONV_FACTOR_DWORDTOREAL;
FlowrateActValueInternal	:=DWORD_TO_REAL(stInputPara.diFlowAct) / CONV_FACTOR_DWORDTOREAL;
DriveDiagnosis                         := stInputPara.dwDriveDiagnosticNumber;


(* Preparing Internal bits / FB output from Signal Status word *)
bModePMActive :=(wSignalStatusWord.1); (*NOT (wSignalStatusWord.1);*)
InStandstill := wSignalStatusWord.3;
bVelCmdValReached := wSignalStatusWord.4;
bDriveHalt := wSignalStatusWord.5;

VelocityLowLevelWarning := wAxisMessages.1;
VelocityHighLimitActive    := wAxisMessages.3;
TorqueHighLimitActive      := wAxisMessages.5;

bMLDPump2OnCmd        := wSignalStatusWord.14;
bMLDRunning                    := wSignalStatusWord.15;

(* Preparing Internal bits / FB output from Process Control Status word *)
bPressureControlActive := wMLDStatusWord.0;
bPressureCmdValReached := wMLDStatusWord.1;
ProcessOutputHLActive := wMLDStatusWord.2;
ProcessOutputLLActive := wMLDStatusWord.3;
ProcessControlError := wMLDStatusWord.4;

(* Reset all bits for Active parameter set number *)
uiActiveParameterSetNoInternal := 0;
(* write bits from MLDStatus words *)
uiActiveParameterSetNoInternal.0 := wMLDStatusWord.14;
uiActiveParameterSetNoInternal.1 := wMLDStatusWord.15;
(* Add 1 because Active set number is ranging from 1..4 for bit value range 00..11 *)
ActiveParameterSetNo := uiActiveParameterSetNoInternal + 1;


(* Preparing Internal bits / FB output from Drive status word*)
bOpModeAck_bit0 := wDriveStatusWord.8;
bOpModeAck_bit1 := wDriveStatusWord.9;
bOpModeAck_bit2 := wDriveStatusWord.10;
bDriveMessageClass3 := wDriveStatusWord.11;
DriveWarning := wDriveStatusWord.12;
DriveError :=  wDriveStatusWord.13;

IF PressureUnit = 1 THEN (* Unit in Percentage of Nominal Value *)
	IF NominalPressureValue <> 0 THEN
		PressureActValue := (PressureActValueInternal / NominalPressureValue) * PERCENTAGE_BASE   ;
	ELSE
		PressureActValue := 0;
	END_IF
ELSE
	PressureActValue := PressureActValueInternal;
END_IF

IF FlowrateUnit = 1 THEN (* Unit in Percentage of Nominal Value *)
	IF NominalFlowrateValue <> 0 THEN
		FlowrateActValue := ( FlowrateActValueInternal  / NominalFlowrateValue) * PERCENTAGE_BASE;

		FlowrateCmdValueInternal := (FlowrateCmdValue * NominalFlowrateValue ) / PERCENTAGE_BASE;
	ELSE
		FlowrateActValue := 0;
		FlowrateCmdValueInternal := 0;
	END_IF
ELSE
	FlowrateActValue := FlowrateActValueInternal;
	FlowrateCmdValueInternal := FlowrateCmdValue ;
END_IF

DriveMode := 0; (* reset all bits *)
DriveMode.0 := wDriveStatusWord.14; (* actualize bit 0 *)
DriveMode.1 := wDriveStatusWord.15; (* actualize bit 1 *)

(* Create Drive State Output *)
IF bModePMActive THEN
	(* Mode PM Active *)
	DriveState := DriveState_Mode_PM;
ELSE
	IF bDriveHalt THEN
		(* 'AH' mode active *)
		DriveState := DriveState_Mode_AH;
	ELSE
		IF (DriveMode = 3) THEN
			IF NOT bMLDRunning THEN
				(* 'AF' mode active *)
				DriveState := DriveState_Mode_AF;
			ELSE
				IF bPressureControlActive THEN
					(* Pressure control mode active *)
					DriveState := DriveState_Mode_PC;
				ELSE
					(* flow rate control mode active *)
					DriveState := DriveState_Mode_FC;
				END_IF
			END_IF
		ELSIF (DriveMode = 2) THEN
			(* Ab' mode active *)
			DriveState := DriveState_Mode_Ab;
		ELSIF	(DriveMode = 1) THEN
			(* 'bb' mode active *)
			DriveState := DriveState_Mode_bb;
		ELSE
			(* Mode Invalid *)
			DriveState := DriveState_Mode_Invalid;
		END_IF
	END_IF
END_IF

(* Mode specific operations and calculations *)
CASE DriveState OF

DriveState_Mode_PC:
(* Pressure Control Mode Active *)
	CommandValueReached := bPressureCmdValReached;
	(* start Pump01 if commanded *)
	Pump01On := PumpOn;

	(* Pump02 is controlled from MLD program *)
	Pump02On := PumpOn AND bMLDPump2OnCmd;

	(* initialize total volume *)
	IF Pump01On THEN
		dwTotalVolume := VolumePump01;
		IF Pump02On THEN
			dwTotalVolume := VolumePump01 + VolumePump02;
		END_IF
	ELSE
		dwTotalVolume := 0;
	END_IF

	IF (dwTotalVolume = 0 ) THEN
		(* reset velocty command, no Volume no flow rate control *)
		diVelocityLimitPos := REAL_TO_DINT(DEFAULT_N_POSITIVE_LIMIT * CONV_FACTOR_REALTODWORD)  ;               (* write default value when Volume is not set  *)
	ELSE
		(* velocty command value is derived by deviding Flowrate Command value with Total volume *)
		diVelocityLimitPos :=REAL_TO_DINT(( FlowrateCmdValueInternal / dwTotalVolume)*CONV_FACTOR_REALTODWORD);
	END_IF

	IF PressureUnit = 1 THEN (* Unit in Percentage of Nominal Value *)
		IF NominalPressureValue <> 0 THEN  (*REAL TO DRIVE UNDERSTANDABLE DWORD*)
			PressureCmdValueInternal := (PressureCmdValue * NominalPressureValue) / (PERCENTAGE_BASE ) ;
		ELSE
			PressureCmdValueInternal := 0;
		END_IF
	ELSE
		PressureCmdValueInternal := PressureCmdValue;
	END_IF

	(* transfer Pressure Command value to drive *)
	diPressureCmd := REAL_TO_DINT (( PressureCmdValueInternal)*CONV_FACTOR_REALTODWORD);

	(* reset velocty command *)
	diVelocityCmd := 0;

DriveState_Mode_FC:
(* Flow rate Control Mode Active *)
	(* Flow rate value reached when Velocity is within tolerance window *)
	CommandValueReached := bVelCmdValReached;
	(* start Pump01 if commanded *)
	Pump01On := PumpOn;
	(* Pump02 is on along with Pump01 *)
	Pump02On := PumpOn ;

	(* reset velocty Limit Value to Default *)
	diVelocityLimitPos := REAL_TO_DINT(DEFAULT_N_POSITIVE_LIMIT*CONV_FACTOR_REALTODWORD);

	(* initialize total volume*)
	IF Pump01On THEN (* and Pump02 is also On *)
		dwTotalVolume := VolumePump01 + VolumePump02;
	ELSE
		dwTotalVolume := 0;
	END_IF

	IF (dwTotalVolume = 0 ) THEN
		(* reset velocty command, no Volume no flow rate control *)
		diVelocityCmd := 0;
	ELSE
		(* velocty command value is derived by deviding Flowrate Command value with Total volume *)
		diVelocityCmd := REAL_TO_DINT((FlowrateCmdValueInternal / dwTotalVolume)*CONV_FACTOR_REALTODWORD);
	END_IF

	(* Pressure Command zero in Flow rate control *)
	diPressureCmd := 0;

ELSE
	(* reset all outputs if not in Process Control mode *)
	dwTotalVolume := 0;
	diVelocityCmd := 0;
	diPressureCmd := 0;
	CommandValueReached := FALSE;
	Pump01On:=FALSE;
	Pump01On:=FALSE;
END_CASE
(* end of Mode specific operations *)

(* set Master control word and Signal control word *)
wMasterControlWord.14 := DriveEnable;
wMasterControlWord.15 := DriveEnable;
wMasterControlWord.13 := DriveStart; (* Drive Halt Command must be set to Activate AF mode at Drive*)

(* reset Diagnostic message using Signal control Word Bit 5 , S144 *)
wSignalControlWord.5 := ResetDriveError;

(* Command for changing the operating mode from Pressure control to Flow rate control and vice versa *)
IF ( OperatingMode = 1)  AND DriveEnable AND DriveStart THEN
	wMLDControlWord.0 := TRUE;
ELSE
	wMLDControlWord.0 := FALSE;
END_IF
(* command to open / close Pump 01 *)
wMLDControlWord.2 := Pump01On;

(* Information to drive about Injection Phase  *)
wMLDControlWord.8 := InjectionPhaseActive;

IF (ParameterSetNo>0) AND(ParameterSetNo<=4)THEN
	uiParameterSetNoInternal := ParameterSetNo  - 1; (* ParameterSetNo = 4  --> bit 15/14 11 in MLDControlword *)
ELSE
	uiParameterSetNoInternal := 0; (* Invalid ParameterSetNo*)
END_IF
(* set PrameterSetNo bits in MLD control word *)
wMLDControlWord.14 := uiParameterSetNoInternal.0;
wMLDControlWord.15 := uiParameterSetNoInternal.1;

(* Transfer Command values to the respective output variables *)
stOutputPara.wMasterControlWord := wMasterControlWord;
stOutputPara.wSignalControlWord:= wSignalControlWord ;
stOutputPara.diVelocityCmd := diVelocityCmd;
stOutputPara.diPressureCmd:= diPressureCmd;
stOutputPara.wProcessControlWord := wMLDControlWord;
stOutputPara.diVelocityLimitPos := diVelocityLimitPos;
stOutputPara.diVolumePump01:=REAL_TO_DWORD(VolumePump01*CONV_FACTOR_VOLUME);
stOutputPara.diVolumePump02:=REAL_TO_DWORD(VolumePump02*CONV_FACTOR_VOLUME);
END_FUNCTION_BLOCK

(* POU FB_Process_Control_using_MUX, ST *)
(*#########################################################################################*)
(* General Header *)
(*----------------------------------------------------------------------------------------------------------------------------------------------------------------*)
(* Short description :		      Function Block "FB_Process_control" controls Process values using MLD program     *)
(* Version : 					      01VRS                                                                                                                                       *)
(* Name : 					      Upendra Chauhan                                                                                                                    *)
(* Date : 					      2012-02-23                                                                                                                               *)
(* Company : 				      Bosch Rexroth AG                                                                                                                    *)
(* Target : 					      >MPx07VRS                                                                                                                             *)
(* Functional description :		The "FB_Process_Control" FUNCTION block provides a user interface for the             *)
(*                                                     Process control FUNCTION block available in the Indradrive using MLD. In addition    *)
(*                                                     to the interface FOR Pressure control, this FB also gives a possibility OF using           *)
(*                                                     Flow rate control instead OF the Pressure control. This FB uses Multiplex channel       *)
(*                                                     (8 Channels) FOR cyclic data communication between Control AND Indradrive            *)
(*----------------------------------------------------------------------------------------------------------------------------------------------------------------*)
(* Handling specials :                                                                                                                                                                      *)
(*----------------------------------------------------------------------------------------------------------------------------------------------------------------*)
(* Additional Header                                                                                                                                                                        *)
(*----------------------------------------------------------------------------------------------------------------------------------------------------------------*)
(* Version : 1.0	                              *)
(* Name : urc2kor ( DC-IA/EDY )   *)
(* Date : 08,05,2012                       *)
(* Company : Bosch Rexroth          *)
(*-----------------------------------------------------------------------------------------------------------------------------------------------------------------*)
(* Version : 1.1	                                                                                                                                                                                           *)
(* Name : urc2kor ( DC-IA/EDY )                                                                                                                                                               *)
(* Date : 29.10.2012                                                                                                                                                                                   *)
(* Company : Bosch Rexroth                                                                                                                                                                      *)
(* Drive Halt Bit activated with DriveStart Input. Without this it is not possible to Activate AF mode at Drive                                   *)
(*--------------------------------------------------------------------------------------------------------------------------------------------------------------------------*)
(* Version : 1.2	                                                                                                                                                                                           *)
(* Name : urc2kor ( DC-IA/EDY )                                                                                                                                                               *)
(* Date : 11.12.2012                                                                                                                                                                                   *)
(* Company : Bosch Rexroth                                                                                                                                                                      *)
(* Drive Halt acknoledgement is configured in SignalStatusWord Bit-5. Bit 3-4 was wrong, corrected the same.                          *)
(* Process control was deactivated when the DriveStart or DriveEnable is removed.                                                                        *)
(*--------------------------------------------------------------------------------------------------------------------------------------------------------------------------*)
(*##########################################################################################*)
(*##########################################################################################*)
FUNCTION_BLOCK FB_Process_Control_using_MUX
VAR_INPUT
	DriveEnable : BOOL;
	DriveStart : BOOL;
	ResetDriveError : BOOL;
	PumpOn : BOOL;
	OperatingMode : INT;
	PressureCmdValue : DINT;
	FlowrateCmdValue : DINT;
	VolumePump01 : DINT;
	VolumePump02 : DINT;
	stInputPara : st_Indradrive_ProcessControl_MUX_input;  (* PD_IN_PROCESS_CONTROL; *)
END_VAR
VAR_OUTPUT
	DriveState : INT;
	InStandstill : BOOL;
	CommandValueReached : BOOL;
	Pump01On : BOOL;
	Pump02On: BOOL;
	VelocityHighLimitActive: BOOL;
	VelocityLowLevelWarning: BOOL;
	TorqueHighLimitActive : BOOL;
	ProcessOutputHLActive : BOOL;
	ProcessOutputLLActive:BOOL;
	ProcessControlError : BOOL;
	DriveWarning: BOOL;
	DriveError: BOOL;
	PressureActValue : DINT;
	FlowrateActValue: DINT;
	DriveDiagnosis : DWORD;
	stOutputPara : st_Indradrive_ProcessControl_MUX_output;  (* EK_OUT_PROCESS_CONTROL; *)
END_VAR
VAR
	wMasterControlWord                   : WORD := 0 ;
	wDriveStatusWord                       : WORD := 0;
	wSignalControlWord                    : WORD := 0 ;
	wSignalStatusWord                     : WORD := 0;

	fbMuxIndradrive                             : FB_Indradrive_MUX_8 ;

	diVelocityAct: DINT := 0;
	wMLDStatusWord: WORD;
	bMLDPump2OnCmd: BOOL := FALSE;
	bMLDRunning: BOOL := FALSE;
	bPressureControlActive: BOOL := FALSE;
	bPressureCmdValReached: BOOL := FALSE;
	bOpModeAck_bit0: BOOL := FALSE;
	bOpModeAck_bit1: BOOL := FALSE;
	bDriveHalt: BOOL := FALSE;
	bModePMActive: BOOL := FALSE;
	bVelCmdValReached: BOOL := FALSE;
	bOpModeAck_bit2: BOOL := FALSE;
	bDriveMessageClass3: BOOL := FALSE;
	DriveMode: WORD := 0;
	dwTotalVolume: DWORD := 0;
	diVelocityCmd: DINT := 0;
	diPressureCmd: DINT := 0;
	wMLDControlWord: WORD := 0;
END_VAR
(* Read Actual values from Drive *)
(* Convert Parameter specific datatypes to DWORD *)
wDriveStatusWord                   := DWORD_TO_WORD (stInputPara.wDriveStatusWord);
wSignalStatusWord                  := DWORD_TO_WORD (fbMuxIndradrive.dwValue_READ_2);
diVelocityAct                             := DWORD_TO_DINT (fbMuxIndradrive.dwValue_READ_3);
DriveDiagnosis                         := fbMuxIndradrive.dwValue_READ_5;
PressureActValue                     := DWORD_TO_DINT (fbMuxIndradrive.dwValue_READ_6);
wMLDStatusWord                    := DWORD_TO_WORD (fbMuxIndradrive.dwValue_READ_7);

(* Preparing Internal bits / FB output from Signal Status word *)
bModePMActive := NOT (wSignalStatusWord.1);
InStandstill := wSignalStatusWord.3;
bVelCmdValReached := wSignalStatusWord.4;
bDriveHalt := wSignalStatusWord.5;

VelocityLowLevelWarning := wSignalStatusWord.11;
VelocityHighLimitActive    := wSignalStatusWord.12;
TorqueHighLimitActive      := wSignalStatusWord.13;
bMLDPump2OnCmd        := wSignalStatusWord.14;
bMLDRunning                    := wSignalStatusWord.15;

(* Preparing Internal bits / FB output from Process Control Status word *)
bPressureControlActive := wMLDStatusWord.0;
bPressureCmdValReached := wMLDStatusWord.1;
ProcessOutputHLActive := wMLDStatusWord.2;
ProcessOutputLLActive := wMLDStatusWord.3;
ProcessControlError := wMLDStatusWord.4;

(* Preparing Internal bits / FB output from Drive status word*)
bOpModeAck_bit0 := wDriveStatusWord.8;
bOpModeAck_bit1 := wDriveStatusWord.9;
bOpModeAck_bit2 := wDriveStatusWord.10;
bDriveMessageClass3 := wDriveStatusWord.11;
DriveWarning := wDriveStatusWord.12;
DriveError :=  wDriveStatusWord.13;

DriveMode := 0; (* reset all bits *)
DriveMode.0 := wDriveStatusWord.14; (* actualize bit 0 *)
DriveMode.1 := wDriveStatusWord.15; (* actualize bit 1 *)

